{attribute 'monitoring' := 'call'}
PROPERTY INTERNAL PosHomeCh : LREAL
GET
PosHomeCh := stLocalSettings.stDynStationSettings[E_St010_Settings.eSt010_Settings_PosHomeCh].fValue;
END_GET
END_PROPERTY

{attribute 'monitoring' := 'call'}
PROPERTY INTERNAL PosWork : LREAL
GET
PosWork := stLocalSettings.stDynStationSettings[E_St010_Settings.eSt010_Settings_PosWork].fValue + // 1. Mitnehmerpos.
	  (OvenSegmentHeight * 
		TRUNC(((P_Plant.TrolleyRackDivision * stSt010IOvenA.iConfirmPosition) + 
		(OvenSegmentHeight - OvenFixPartHeight - 50))/OvenSegmentHeight)); // -50 => height axis z
END_GET
END_PROPERTY

{attribute 'monitoring' := 'call'}
PROPERTY INTERNAL PosWorkCh : LREAL
GET
PosWorkCh := stLocalSettings.stDynStationSettings[E_St010_Settings.eSt010_Settings_PosWorkCh].fValue;
END_GET
END_PROPERTY

{attribute 'monitoring' := 'call'}
PROPERTY INTERNAL PosWorkOpn : LREAL
GET
PosWorkOpn := PosWork + 

			  LMOD(((P_Plant.TrolleyRackDivision * stSt010IOvenA.iConfirmPosition) + (P_Plant.TrolleyRackOriginX - OvenFixPartHeight - 50)), 
					OvenSegmentHeight) + 
					50 + // -50 => height axis z
			  P_Plant.TrolleyRackDivision; // ( + TrolleyDevisionY --> safety distance)
END_GET
END_PROPERTY

/// Reset station logic
{attribute 'object_name' := 'Reset'}
METHOD Reset
VAR
END_VAR
// base logic run
SUPER^.Reset();

// reset objects
//diContinuesNok := 0;

IF fbAxis.bError OR NOT RunCycle THEN
	fbAxis.Reset();
END_IF
IF fbAxisCh1.bError OR NOT RunCycle THEN
	fbAxisCh1.Reset();
END_IF
IF fbAxisCh2.bError OR NOT RunCycle THEN
	fbAxisCh2.Reset();
END_IF
END_METHOD

{attribute 'monitoring' := 'call'}
PROPERTY PRIVATE WorkSpeed : LREAL
GET
WorkSpeed := stLocalSettings.stDynStationSettings[E_St010_Settings.eSt010_Settings_WorkSpeed].fValue;
END_GET
END_PROPERTY

{attribute 'monitoring' := 'call'}
PROPERTY PRIVATE WorkSpeedCh : LREAL
GET
WorkSpeedCh := stLocalSettings.stDynStationSettings[E_St010_Settings.eSt010_Settings_WorkSpeedCh].fValue;
END_GET
END_PROPERTY

END_FUNCTION_BLOCK

// ---- POUs/Components/AxisDriver/FB_Axis_Ui.TcPOU
/// Visu Interface für Achse
FUNCTION_BLOCK FB_Axis_Ui EXTENDS FB_ManualUiBase
VAR_INPUT
	///	Zus. Freigabe für Positive Richtung	
	bFreigabe_P		: BOOL := TRUE;
	///	Zus. Freigabe für Negative Richtung	
	bFreigabe_N		: BOOL := TRUE;
	
	/// Tippen +
	bJogP			:BOOL;
	/// Tippen -
	bJogN			:BOOL;
	/// GoTo
	//bGoTo		:BOOL;
	/// Geschwindigkeit
	fVelocity		:REAL := 1;
	
	/// Maximaler Weg pro Bewegung
	fMaxWeg			: REAL := 500;
	bModulo			: BOOL := FALSE;
	bEnableRefReset	: BOOL;	
	bEnableGear		: BOOL := FALSE;
	fGearRatio		: LREAL := 1;
	eMasterAxisId	: E_Axis := E_Axis.eAxis_none;
	bEnableBrakeControl	: BOOL := FALSE;
	bEnableSetPos	: BOOL := FALSE;
	
	// axis manager
	stAxisManager	: ST_AxisManager;
	stUnit			: ST_Text;
END_VAR
VAR_IN_OUT
	/// Achse in GRST
	bInHome			: BOOL;
	// axis reference
	fbAxis			: FB_AxisDriver;
	// hmi control IN
	stHMIControlIn	: ST_HMI_MANUAL_AXIS_IN;
	// hmi control OUT
	stHMIControlOut	: ST_HMI_MANUAL_AXIS_OUT;
END_VAR
VAR_OUTPUT	
	/// 0=Undefiniert; 
	/// 1=Fehler; 
	/// 2=Fahrt Positiv; 
	/// 3=Fahrt Negativ
	/// 4=Stillstand
	/// 5=Synchron
	iStatus				: INT;
	stState				: ST_Text;
	
	/// Servo Istposition
	fPosition			: LREAL;
	diColor_Position	: UDINT := STATICS.stColor.Gray;
	diColor_State		: UDINT;
	diColorSelectedItem	: UDINT;
	sText_State			: STRING;
END_VAR
VAR
	nn	: INT;
	stAxisState				: Tc2_MC2.ST_AxisStatus;
	eManualMode				: E_ManualMode;
	eManualModeOLD			: E_ManualMode;
	
	posEnableManual			: R_TRIG;
	negEnableManual			: F_TRIG;
	posIndexChanged			: R_TRIG;
	rtrigGearIn				: R_TRIG;
	ftrigGearOut			: F_TRIG;
	posGoTo,
	posGear,
	posTip_P,
	posTip_N,
	posRefReset,	
	rtrigTargetListClick,			
	rtrigBrake				: R_TRIG;
	
	fTargetPos				: LREAL;
	fStartPos				: LREAL;
	bManualModeAbsolute,
	bMovingAbs				: BOOL;
	bGear					: BOOL;
	
	bBrakeOff				: BOOL;
	
	posSelGoTo,
	posTippPos,
	posTippNeg,
	posSelJogTipp,
	posSelJog001,
	posSelJog01,
	posSelJog1,
	posSelJog10,
	posSelJog100,
	posSelMoveSollposAbs	: R_TRIG;
	
	tonRefReset				: TON;
	
	fSollPositionLatched	: REAL;
	
	stHomeParameter			: ST_AxisHomingParameter;
	
	tonTagetListClick		: ton;
	bTagetListClickSave		: BOOL;
	nTargetListIdx			: UINT;
	bFromTargetList			: BOOL; // FALSE from Input feld TRUE from List
	
	// master axis reference, if needed (else, set to dummy)
	stMasterAxisRef			: REFERENCE TO AXIS_REF REF= NcIO.stAxisDummy;
END_VAR
VAR PERSISTENT
	stTargetList			: ARRAY[0..9] OF ST_UserControl_Manual_Axis_Item; /// product data
	bCalibratedLocal		: BOOL;
END_VAR

(*
	Baustein zum bedienen einer Achse ueber die Visu
*)
stName := fbAxis.Name;
nTargetListIdx := stHMIControlIn.nSelectedRowIndex;
M_AxisManager();

IF (diObjectIndex = diSelectedObjectIndex) AND (diObjectIndex <> 0) AND bEnableManual THEN
	bManualActive := TRUE;
	stHMIControlOut.bVisible := TRUE;
	stHMIControlOut.bVisibleGear := bEnableGear;
	stHMIControlOut.bVisibleRefReset := bEnableRefReset;
	stHMIControlOut.bVisibleBrake := bEnableBrakeControl;
	stHMIControlOut.bVisibleSetPos := bEnableSetPos;
	stName:= stHMIControlOut.stObjectName := fbAxis.Name;

	stHMIControlOut.sOverride := SEL(fbAxis.bHoldActiv,LREAL_TO_FMTSTR(REAL_TO_LREAL(fbAxis.Override), 4, FALSE),'Hold Activ');
	stHMIControlOut.sTargetPosition := LREAL_TO_FMTSTR(REAL_TO_LREAL(fTargetPos), 4, FALSE);
	
	IF bModulo THEN
		stHMIControlOut.sActPosition := LREAL_TO_FMTSTR(fbAxis.ModuloPosition, 4, FALSE);
	ELSE
		stHMIControlOut.sActPosition := LREAL_TO_FMTSTR(fbAxis.Position, 4, FALSE);
	END_IF
	
	IF stAxisState.Coupled THEN
		stHMIControlOut.stGearStatus := F_CreateDynText("coupled", 0);
	ELSE
		stHMIControlOut.stGearStatus := F_CreateDynText("uncoupled", 0);
	END_IF
	
	IF NOT fbAxis.Homed THEN
		stHMIControlOut.stRefStatus := F_CreateDynText("unreferenced", 0);
	ELSE
		stHMIControlOut.stRefStatus := F_CreateDynText("referenced", 0);
	END_IF
	
	stHMIControlOut.stButtonGoTo.stName := CONST.stTextListGlobal.stText_GoTo;
	stHMIControlOut.stButtonJogPos.stName := CONST.stTextListGlobal.stText_JogPos;
	stHMIControlOut.stButtonJogNeg.stName := CONST.stTextListGlobal.stText_JogNeg;
	stHMIControlOut.stButtonGear.stName := CONST.stTextListGlobal.stText_Gear;
	stHMIControlOut.stButtonRefReset.stName := CONST.stTextListGlobal.stText_RefReset;
	stHMIControlOut.stButtonBrake.stName := CONST.stTextListGlobal.stText_Brake;
	stHMIControlOut.stButtonSetPos.stName := CONST.stTextListGlobal.stText_SetPos;

	stHMIControlOut.aJogModeName[0] :=  CONST.stTextListGlobal.stText_Jogpermanent;
	stHMIControlOut.aJogModeName[1] :=  CONST.stTextListGlobal.stText_Jog_0_01;
	stHMIControlOut.aJogModeName[2] :=  CONST.stTextListGlobal.stText_Jog_0_1;
	stHMIControlOut.aJogModeName[3] :=  CONST.stTextListGlobal.stText_Jog_1_0;	
	stHMIControlOut.aJogModeName[4] :=  CONST.stTextListGlobal.stText_Jog_10_0;	
	
	stHMIControlOut.stButtonGoTo.stColor.color := F_ColorToStringHexColor(STATICS.stColor.Theme);
	stHMIControlOut.stButtonJogPos.stColor.color := F_ColorToStringHexColor(STATICS.stColor.Theme);
	stHMIControlOut.stButtonJogNeg.stColor.color := F_ColorToStringHexColor(STATICS.stColor.Theme);
	stHMIControlOut.stButtonGear.stColor.color := F_ColorToStringHexColor(STATICS.stColor.Theme);
	stHMIControlOut.stButtonRefReset.stColor.color := F_ColorToStringHexColor(STATICS.stColor.Theme);
	stHMIControlOut.stButtonBrake.stColor.color := F_ColorToStringHexColor(STATICS.stColor.Theme);
	
	IF stHMIControlIn.stButtonGoTo.bClick AND bMovingAbs THEN
		stHMIControlOut.stButtonGoTo.stColor.color := F_ColorToStringHexColor(STATICS.stColor.LimeGreen);
	END_IF
	IF stHMIControlIn.stButtonJogPos.bClick AND NOT bMovingAbs AND fbAxis.Velocity > 0.5 THEN
		stHMIControlOut.stButtonJogPos.stColor.color := F_ColorToStringHexColor(STATICS.stColor.LimeGreen);
	END_IF
	IF stHMIControlIn.stButtonJogNeg.bClick AND NOT bMovingAbs AND fbAxis.Velocity < -0.5 THEN
		stHMIControlOut.stButtonJogNeg.stColor.color := F_ColorToStringHexColor(STATICS.stColor.LimeGreen);
	END_IF
	IF bGear THEN
		stHMIControlOut.stButtonGear.stColor.color := F_ColorToStringHexColor(STATICS.stColor.LimeGreen);
	END_IF
	IF tonRefReset.Q THEN
		stHMIControlOut.stButtonRefReset.stColor.color := F_ColorToStringHexColor(STATICS.stColor.LimeGreen);
	END_IF	
	IF bBrakeOff THEN
		stHMIControlOut.stButtonBrake.stColor.color := F_ColorToStringHexColor(STATICS.stColor.LimeGreen);
	END_IF	

	// Timer, Flanken
	posTip_P(CLK := bJogP OR stHMIControlIn.stButtonJogPos.bClick);
	posTip_N(CLK := bJogN OR stHMIControlIn.stButtonJogNeg.bClick);
	posGoTo(CLK := (*bGoTo OR*) stHMIControlIn.stButtonGoTo.bClick);
	posGear(CLK := stHMIControlIn.stButtonGear.bClick);
	rtrigTargetListClick(CLK := stHMIControlIn.bSetTargetFromList);
	tonRefReset.PT := T#1S;
	tonRefReset.IN := stHMIControlIn.stButtonRefReset.bClick;
	tonRefReset();
	posRefReset(CLK := tonRefReset.Q);	
	rtrigBrake(CLK := stHMIControlIn.stButtonBrake.bClick); 
	IF posTip_N.Q OR posTip_P.Q THEN
		bMovingAbs := FALSE;
		bManualModeAbsolute := FALSE;
	ELSIF posGoTo.Q THEN
		bManualModeAbsolute := TRUE;
	END_IF
	IF posGear.Q AND fbAxis.NotMoving THEN
		bGear := NOT bGear;
	END_IF
	IF rtrigBrake.Q AND (fbAxis.NotMoving OR TRUE)THEN
		bBrakeOff := NOT bBrakeOff;
	END_IF
ELSE
	IF bManualActive THEN
		bManualActive := FALSE;
		stHMIControlOut.bVisible := FALSE;
	END_IF
	bBrakeOff := FALSE;
END_IF	
	
// nicht aktiv -> alles löschen und Exit
IF NOT fbAxis.Active THEN
	bError := FALSE ;
	stErrorText := CONST.stTextListGlobal.stText_notext;
	iStatus := 0;// 0=Undefiniert
	fPosition := 0;
	A_StateMapping();
	RETURN;
END_IF

// Object mit Index ausgewählt
IF (diObjectIndex = diSelectedObjectIndex) THEN
	diColorSelectedItem := STATICS.stColor.LimeGreen;
ELSE
	diColorSelectedItem := STATICS.stColor.Gray;
END_IF

bError := fbAxis.State = E_ComponentState.eComponentState_error;
IF bError THEN
	stErrorText := F_CreateDynTextDefault(fbAxis.ClearText);
ELSE
	stErrorText := CONST.stTextListGlobal.stText_notext;
END_IF
fPosition := fbAxis.Position; // Istposition der Achse

// Status
stAxisState := fbAxis.AxisState;
IF bError THEN
	iStatus := 1; // 1=Fehler; 
	diColor_State:= STATICS.stColor.Red;
	stState.wsNameId := "error";
	stState.wsName := "error";
	stState.nNameId :=1;
ELSIF stAxisState.Moving AND stAxisState.PositiveDirection THEN
	iStatus := 2; // 2=Fahrt Positiv; 
	diColor_State:= STATICS.stColor.Green;
	stState.wsNameId := "movepositive";
	stState.wsName := "movepositive";
	stState.nNameId :=2;
ELSIF stAxisState.Moving AND stAxisState.NegativeDirection THEN
	iStatus := 3; // 3=Fahrt Negativ;
	diColor_State:= STATICS.stColor.Green;
	stState.wsNameId := "movenegative";
	stState.wsName := "movenegative";
	stState.nNameId :=3;
ELSIF stAxisState.Coupled THEN
	iStatus := 5; // 5=Synchron
	diColor_State:= STATICS.stColor.LightSkyBlue;
	stState.wsNameId := "coupled";
	stState.wsName := "coupled";
	stState.nNameId :=5;
ELSIF NOT stAxisState.Moving THEN
	iStatus := 4; // 4=Stillstand
	diColor_State:= STATICS.stColor.Gray;
	stState.wsNameId := "notmoveing";
	stState.wsName := "notmoveing";
	stState.nNameId :=4;
ELSE
	iStatus := 0;// 0=Undefiniert
	diColor_State:= STATICS.stColor.Orange;
	stState.wsNameId := "undifined";
	stState.wsName := "undifined";
	stState.nNameId :=0;
END_IF

//Statuszahl Text Zuweisung
CASE iStatus OF
	0:
		sText_State := ('Undefiniert');
	1:
		sText_State := ('Fehler');
	2:
		sText_State := ('Fahrt Positiv');
	3:
		sText_State := ('Fahrt Negativ');
	4:
		sText_State := ('Stillstand OK');
	5:
		sText_State := ('Synchron');
END_CASE

bWarning := FALSE;
stWarnText := CONST.stTextListGlobal.stText_notext;

// Achse stoppen bei Umschaltung(en)
posEnableManual(CLK := bEnableManual);
negEnableManual(CLK := bEnableManual);
posIndexChanged(CLK := bEnableManual AND (diObjectIndex <> diSelectedObjectIndex));
IF posEnableManual.Q OR negEnableManual.Q OR posIndexChanged.Q THEN
	IF fbAxis.Moving THEN
		fbAxis.Halt();
	END_IF
	bMovingAbs := FALSE;
END_IF

// Homing Zurücksetzen
IF posRefReset.Q AND fbAxis.NotMoving AND fbAxis.Homed AND bEnableRefReset THEN
	stHomeParameter.eHomingMode := MC_HomingMode.MC_ResetCalibration;
	fbAxis.HomeEx(stHomeParameter);
END_IF

// exit wenn nicht dieses Objekt
IF NOT bEnableManual OR (diObjectIndex <> diSelectedObjectIndex) THEN
	bMovingAbs := FALSE;
	A_StateMapping();
	RETURN;
END_IF


// Handbedienlogik
// werwenden von Handbediencontrol direkt
// Status wird in diesem FB gemerkt und wiedereingestellt

// Auswahl Manuelle Funktionen
A_SelectManualMode();

// Modus wurde geändert -> Achse stoppen
IF eManualMode <> eManualModeOLD THEN
	eManualModeOLD := eManualMode;
	IF fbAxis.Moving THEN
		fbAxis.Halt();
	END_IF
	bMovingAbs := FALSE;
	bBrakeOff := FALSE;
END_IF

// Bei Stillstand und Taste Gear in HMI Koppeln
rtrigGearIn(CLK := bGear);
ftrigGearOut(CLK := bGear);
IF fbAxis.NotMoving AND rtrigGearIn.Q AND bEnableGear THEN
	fbAxis.GearIn(fGearRatio, eMasterAxisId, stMasterAxisRef);
END_IF
IF fbAxis.NotMoving AND ftrigGearOut.Q THEN
	fbAxis.GearOut();
END_IF

//Bremsen Steuerung
IF fbAxis.bHasJob OR NOT bEnableBrakeControl THEN
	bBrakeOff := FALSE;
END_IF
IF bBrakeOff THEN
	; //todo brake control
END_IF

FOR nn := 0 TO 9 DO
	stHMIControlout.stTargetList[nn].stName := stTargetList[nn].stName;
	stHMIControlout.stTargetList[nn].stPos.wsNameId := stHMIControlout.stTargetList[nn].stPos.wsName := TO_WSTRING(stTargetList[nn].fPos);
END_FOR

//set Target from Target List
fTargetPos := SEL(bFromTargetList AND nTargetListIdx >= 0 AND nTargetListIdx <= 9, 
					stHMIControlIn.fTargetPosition, 
					stTargetList[nTargetListIdx].fPos);

IF rtrigTargetListClick.Q THEN
	bTagetListClickSave := TRUE;
END_IF

tonTagetListClick(IN := bTagetListClickSave, PT := T#1S);
IF tonTagetListClick.Q THEN
	bTagetListClickSave := FALSE;
	IF (stTargetList[nTargetListIdx].stName.wsNameId <> "") OR (stTargetList[nTargetListIdx].stName.wsName <> "") THEN
		bFromTargetList := TRUE;
	END_IF
END_IF
IF stHMIControlIn.bSetTarget THEN
	bFromTargetList := FALSE;	
END_IF

// Manuelle Bewegungen
// Tippen konstant
IF (eManualMode = E_ManualMode.eManualMode_Tippen) THEN
	IF posTip_P.Q OR posTip_N.Q THEN
		bInHome := FALSE;
		fStartPos := fbAxis.Position;
	END_IF
	fbAxis.JogExVel(((bJogN OR stHMIControlIn.stButtonJogNeg.bClick) AND bFreigabe_N), 	// Tip N, max Weg		ABS(fbAxis.Position - fStartPos) < fMaxWeg
					((bJogP OR stHMIControlIn.stButtonJogPos.bClick) AND bFreigabe_P), 	// Tip P, max Weg		ABS(fbAxis.Position - fStartPos) < fMaxWeg)
					fVelocity/2, E_JogMode.MC_JOGMODE_CONTINOUS);
					
// Tippen um 0.01 Einheit
ELSIF (eManualMode = E_ManualMode.eManualMode_Jog001) THEN
	IF posTip_P.Q AND bFreigabe_P THEN
		bInHome := FALSE;
		fbAxis.MoveRelExVel(0.01, fVelocity);
	END_IF
	IF posTip_N.Q AND bFreigabe_N THEN
		bInHome := FALSE;
		fbAxis.MoveRelExVel(-0.01, fVelocity);
	END_IF					

// Tippen um 0.1 Einheit
ELSIF (eManualMode = E_ManualMode.eManualMode_Jog01) THEN
	IF posTip_P.Q AND bFreigabe_P THEN
		bInHome := FALSE;
		fbAxis.MoveRelExVel(0.1, fVelocity);
	END_IF
	IF posTip_N.Q AND bFreigabe_N THEN
		bInHome := FALSE;
		fbAxis.MoveRelExVel(-0.1, fVelocity);
	END_IF

// Tippen um 1 Einheit
ELSIF (eManualMode = E_ManualMode.eManualMode_Jog1) THEN
	IF posTip_P.Q AND bFreigabe_P THEN
		bInHome := FALSE;
		fbAxis.MoveRelExVel(1.0, fVelocity);
	END_IF
	IF posTip_N.Q AND bFreigabe_N THEN
		bInHome := FALSE;
		fbAxis.MoveRelExVel(-1.0, fVelocity);
	END_IF

// Tippen um 10 Einheiten
ELSIF (eManualMode = E_ManualMode.eManualMode_Jog10) THEN
	IF posTip_P.Q AND bFreigabe_P THEN
		bInHome := FALSE;
		fbAxis.MoveRelExVel(10.0, fVelocity);
	END_IF
	IF posTip_N.Q AND bFreigabe_N THEN
		bInHome := FALSE;
		fbAxis.MoveRelExVel(-10.0, fVelocity);
	END_IF

// Tippen um 100 Einheiten
(*ELSIF (eManualMode = E_ManualMode.eManualMode_Jog100) THEN
	IF posTip_P.Q AND bFreigabe_P THEN
		fbAxis.MoveRelExVel(100.0, fVelocity);
	END_IF
	IF posTip_N.Q AND bFreigabe_N THEN
		fbAxis.MoveRelExVel(-100.0, fVelocity);
	END_IF	*)
END_IF

// Position anfahren solange Tip Taste gedrueckt
IF bManualModeAbsolute THEN //IF (eManualMode = E_ManualMode.eManualMode_MoveSollAbs) THEN

	// Halt	
	IF NOT stHMIControlIn.stButtonGoTo.bClick THEN//bGoTo THEN
		IF fbAxis.Moving THEN
			fbAxis.Halt();
		END_IF
		fSollPositionLatched := fTargetPos;//stVisuControlPanel.fSollPosition;
		bMovingAbs := FALSE;
		
	// los
	// Start oder Soll Position geändert
	ELSIF posGoTo.Q OR (fbAxis.Moving AND fSollPositionLatched <> fTargetPos(*stVisuControlPanel.fSollPosition*)) THEN
		fSollPositionLatched := fTargetPos;//stVisuControlPanel.fSollPosition;
		fStartPos := fbAxis.Position;
		bMovingAbs := TRUE;
		
		// möchte in Positive Richtung fahren, keine Freigabe = Alarm
		IF ((*stVisuControlPanel.fSollPosition*)fTargetPos > fbAxis.Position) THEN
			IF bFreigabe_P THEN
				IF NOT bModulo THEN
					fbAxis.MoveAbsExVel(fTargetPos(*stVisuControlPanel.fSollPosition*), fVelocity);
				ELSE
					fbAxis.MoveModExVel(fTargetPos(*stVisuControlPanel.fSollPosition*), fVelocity);
				END_IF
				bInHome := FALSE;
			ELSE
				bWarning := TRUE;
				stWarnText := CONST.stTextListGlobal.stText_Comp.stText_AxisUi_PosDirectionWarn;				
			END_IF
			
		// möchte in Negative Richtung fahren, keine Freigabe = Alarm
		ELSIF ((*stVisuControlPanel.fSollPosition*)fTargetPos < fbAxis.Position) THEN
			IF bFreigabe_N THEN
				IF NOT bModulo THEN
					fbAxis.MoveAbsExVel(fTargetPos(*stVisuControlPanel.fSollPosition*), fVelocity);	
				ELSE
					fbAxis.MoveModExVel(fTargetPos(*stVisuControlPanel.fSollPosition*), fVelocity);	
				END_IF		
				bInHome := FALSE;
			ELSE
				bWarning := TRUE;
				stWarnText := CONST.stTextListGlobal.stText_Comp.stText_AxisUi_NegDirectionWarn;				
			END_IF
			
		END_IF
		
	// max. Weg Begrenzen
	ELSIF (ABS(fbAxis.Position - fStartPos) > fMaxWeg) AND fbAxis.Moving AND bMovingAbs THEN
		fbAxis.Halt();
		bMovingAbs := FALSE;
	END_IF
	
END_IF


//IF (eManualMode <> E_ManualMode.eManualMode_MoveSollAbs) THEN
//	bMovingAbs := FALSE;
//END_IF

A_StateMapping();

ACTION A_SelectManualMode:

// Auswahl Manuelle Funktionen

posSelGoTo(CLK := stHMIControlIn.stButtonGoTo.bClick);
posTippPos(CLK := stHMIControlIn.stButtonJogPos.bClick);
posTippNeg(CLK := stHMIControlIn.stButtonJogNeg.bClick);

CASE stHMIControlIn.eJogMode OF
	E_Axis_JogMode.eJogMode_0: // Tippen um Schritt
		eManualMode := E_ManualMode.eManualMode_Tippen;
	E_Axis_JogMode.eJogMode_1: // Tippen um 0,01
		eManualMode := E_ManualMode.eManualMode_Jog001;
	E_Axis_JogMode.eJogMode_2: // Tippen um 0,1
		eManualMode := E_ManualMode.eManualMode_Jog01;
	E_Axis_JogMode.eJogMode_3: // Tippen um 1
		eManualMode := E_ManualMode.eManualMode_Jog1;
	E_Axis_JogMode.eJogMode_4: // Tippen um 10
		eManualMode := E_ManualMode.eManualMode_Jog10;
	E_Axis_JogMode.eJogMode_5: // Tippen um 100
		eManualMode := E_ManualMode.eManualMode_Jog100;
	//E_Axis_JogMode.eJogMode_1: // Absolut Positionieren
	//	eManualMode := E_ManualMode.eManualMode_MoveSollAbs;	
END_CASE

//posSelJogTipp(CLK := stVisuControlPanel.bTippen);
//posSelJog001(CLK := stVisuControlPanel.bJog001);
//posSelJog01(CLK := stVisuControlPanel.bJog01);
//posSelJog1(CLK := stVisuControlPanel.bJog1);
//posSelJog10(CLK := stVisuControlPanel.bJog10);
//posSelJog100(CLK := stVisuControlPanel.bJog100);
//posSelMoveSollposAbs(CLK := stVisuControlPanel.bSollposAnfahren);

//IF posSelJogTipp.Q THEN
//	eManualMode := E_ManualMode.eManualMode_Tippen;
//END_IF
//IF posSelJog001.Q THEN
//	eManualMode := E_ManualMode.eManualMode_Jog001;
//END_IF
//IF posSelJog01.Q THEN
//	eManualMode := E_ManualMode.eManualMode_Jog01;
//END_IF
//IF posSelJog1.Q THEN
//	eManualMode := E_ManualMode.eManualMode_Jog1;
//END_IF
//IF posSelJog10.Q THEN
//	eManualMode := E_ManualMode.eManualMode_Jog10;
//END_IF
//IF posSelJog100.Q THEN
//	eManualMode := E_ManualMode.eManualMode_Jog100;
//END_IF
//IF posSelMoveSollposAbs.Q THEN
//	eManualMode := E_ManualMode.eManualMode_MoveSollAbs;
//END_IF

//// andere Typen
//stVisuControlPanelStatus.bAusSelected := FALSE;
//stVisuControlPanelStatus.bEinSelected := FALSE;
//// Servos
/////Servo Tippen	
//stVisuControlPanelStatus.bTippenSelected := (eManualMode = E_ManualMode.eManualMode_Tippen);
/////Servo Jog 0.01
//stVisuControlPanelStatus.bJog001Selected := (eManualMode = E_ManualMode.eManualMode_Jog001);
/////Servo Jog 0.1
//stVisuControlPanelStatus.bJog01Selected := (eManualMode = E_ManualMode.eManualMode_Jog01);
/////Servo Jog 1
//stVisuControlPanelStatus.bJog1Selected := (eManualMode = E_ManualMode.eManualMode_Jog1);
/////Servo Jog 10
//stVisuControlPanelStatus.bJog10Selected := (eManualMode = E_ManualMode.eManualMode_Jog10);
/////Servo Jog 100
//stVisuControlPanelStatus.bJog100Selected := (eManualMode = E_ManualMode.eManualMode_Jog100);
/////Servo Sollposition Anfahren
//stVisuControlPanelStatus.bSollposAnfahrenSelected := (eManualMode = E_ManualMode.eManualMode_MoveSollAbs);
END_ACTION

ACTION A_StateMapping:
IF NOT __ISVALIDREF(stStateObject) THEN
	RETURN;
END_IF

// state mapping
stStateObject.stState := stState;
stStateObject.stValue.wsName := TO_WSTRING(LREAL_TO_FMTSTR(REAL_TO_LREAL(fPosition), 2, FALSE));
stStateObject.nIndexColor := diColorSelectedItem;
END_ACTION

METHOD PRIVATE M_AxisManager : BOOL
VAR_INPUT
END_VAR
// map axis info
stAxisManager.bAxisEnabled := fbAxis.bEnable;
stAxisManager.bCalibrated := SEL(stAxisManager.bUseLocalCalibration, fbAxis.Homed, bCalibratedLocal);
stAxisManager.fActPos := fbAxis.Position;
stAxisManager.stBmk := stBmk;
stAxisManager.stName := stName;
stAxisManager.stUnit := stUnit;
//stAxisManager.stInfo := ST_Text;

// set/reset calibration
IF stAxisManager.bSetCalibration THEN
	stAxisManager.bSetCalibration := FALSE;
	IF stAxisManager.bUseLocalCalibration THEN bCalibratedLocal := TRUE; RETURN; END_IF
	fbAxis.SetCalibration(TRUE);
ELSIF stAxisManager.bResetCalibration THEN
	stAxisManager.bResetCalibration := FALSE;
	IF stAxisManager.bUseLocalCalibration THEN bCalibratedLocal := FALSE; RETURN; END_IF
	fbAxis.SetCalibration(FALSE);
END_IF

// set ax pos offset
IF stAxisManager.bSetPosGo THEN
	stAxisManager.bSetPosGo := FALSE;
	fbAxis.SetAxPosOffs(stAxisManager.fSetPos);
END_IF
END_METHOD

METHOD PUBLIC M_SetMaserAxRef : BOOL
VAR_IN_OUT
	fbAxRef : AXIS_REF;
END_VAR
stMasterAxisRef REF= fbAxRef;
END_METHOD

METHOD PUBLIC M_TargetListAddItem : BOOL
VAR_INPUT
	stSetName		: ST_Text;
	fSetPosition	: LREAL;
END_VAR
FOR nn := 0 TO 9 DO
	IF (stTargetList[nn].stName.wsNameId = stSetName.wsNameId)OR (stTargetList[nn].stName.wsName = stSetName.wsName)THEN
		stTargetList[nn].fPos := fSetPosition;
		EXIT;
	ELSIF (stTargetList[nn].stName.wsNameId = "") AND (stTargetList[nn].stName.wsName = "") THEN
		stTargetList[nn].stName := stSetName;
		stTargetList[nn].fPos := fSetPosition;
		EXIT;
	END_IF
END_FOR
END_METHOD

METHOD M_TargetListClear : BOOL
VAR_INPUT
END_VAR
MEMSET(ADR(stTargetList), 0, SIZEOF(stTargetList));
END_METHOD

PROPERTY ManualMode : E_ManualMode
GET
ManualMode := eManualMode;
END_GET
SET
eManualMode := ManualMode;
END_SET
END_PROPERTY

END_FUNCTION_BLOCK

// ---- POUs/Components/FurnaceDriver/FB_FurnaceDriver.TcPOU
/// Exhaustion driver.
FUNCTION_BLOCK FB_FurnaceDriver EXTENDS FB_ComponentBase

VAR CONSTANT
	nFurnanceScheduleItems		: INT := 7;
END_VAR

VAR
	/// IO structure
	stIn 				: REFERENCE TO ST_FurnaceIn;
	stOut 				: REFERENCE TO ST_FurnaceOut;
	
	/// fb
	fbTmpCtrl			: FB_CTRL_TempController;
	
	/// Sequences
	eSequenceId			: E_FurnaceSeq;
	
	nStep				: INT;
	
	// private var's
	stCTRLParameter		: ST_CTRL_TempCtrlParameter;
	stPIDParameter		: ST_CTRL_ParaController;
	
	fTemperature		: LREAL;
	fSlope				: LREAL;
	fInitial			: LREAL;
	bkpAlarmSupp		: DWORD;	
	eCTRL_Mode 			: E_CTRL_MODE := E_CTRL_MODE.eCTRL_MODE_IDLE; 	(*   eCTRL_MODE_TUNE  ;*)
	bTuned				: BOOL;	
	rtOverheat			: R_TRIG;

END_VAR

///
/// Furnace driver.
/// Hannes Fuger / asma.at / 12.2015
///

METHOD PRIVATE _AUTO 
VAR_INPUT
END_VAR
CASE nStep OF
	
0	:	// switch to Active mode
		eCTRL_Mode := E_CTRL_MODE.eCTRL_MODE_ACTIVE;
		stCtrlParameter.bSelCtrlParameterSet := TRUE;
						
		IF fbTmpCtrl.eCtrlState = e_Ctrl_state.eCTRL_STATE_ACTIVE THEN
			nStep := 99;
		END_IF			


END_CASE
END_METHOD

METHOD _HAND
VAR_INPUT
END_VAR
CASE nStep OF
	
0	:	// switch to Active mode
		eCTRL_Mode := E_CTRL_MODE.eCTRL_MODE_MANUAL;
		stCtrlParameter.bSelCtrlParameterSet := TRUE;
							
		IF fbTmpCtrl.eCtrlState = e_Ctrl_state.eCTRL_STATE_MANUAL THEN
			nStep := 99;
		END_IF	
		
END_CASE
END_METHOD

METHOD _OFF
VAR_INPUT
END_VAR
CASE nStep OF
	
0	:	// switch to Active mode
		eCTRL_Mode := E_CTRL_MODE.eCTRL_MODE_IDLE;
							
		IF fbTmpCtrl.eCtrlState = e_Ctrl_state.eCTRL_STATE_IDLE THEN
			nStep := 99;
		END_IF	
			
END_CASE
END_METHOD

METHOD _TUNE
VAR_INPUT
END_VAR
CASE nStep OF
	
0	:	// switch to Tune mode
		eCTRL_Mode := E_CTRL_MODE.eCTRL_MODE_TUNE;
		// Alarme ausstellen
		bkpAlarmSupp := stCTRLParameter.dwAlarmSupp;
		stCtrlParameter.bSelCtrlParameterSet := FALSE;
		
		IF fbTmpCtrl.eCtrlState = e_Ctrl_state.eCTRL_STATE_TUNING THEN
			nStep := 10;
		END_IF

10	:	IF fbTmpCtrl.eCtrlState = e_Ctrl_state.eCTRL_STATE_TUNED THEN
			nStep := 20;
		END_IF
			
20	:	stPIDParameter := fbTmpCtrl.sParaControllerInternal;
		stCtrlParameter.bSelCtrlParameterSet := TRUE;
		fbTmpCtrl.eCtrlMode := E_CTRL_MODE.eCTRL_MODE_PASSIVE;
		eSequenceId := eFurnaceSeq_none;
		

END_CASE
END_METHOD

PROPERTY CtrlParameter : REFERENCE TO ST_CTRL_TempCtrlParameter
GET
ctrlParameter REF= stCTRLParameter;
END_GET
SET
stCTRLParameter := ctrlParameter;
END_SET
END_PROPERTY

PROPERTY CtrlState : E_CTRL_STATE
GET
CtrlState := fbTmpCtrl.eCtrlState;
END_GET
END_PROPERTY

PROPERTY Error : BOOL
GET
Error := fbTmpCtrl.bError;
END_GET
END_PROPERTY

PROPERTY ErrorId : E_CTRL_ERRORCODES
GET
ErrorId := fbTmpCtrl.eErrorId;
END_GET
END_PROPERTY

METHOD FB_init : BOOL
VAR_INPUT
	bInitRetains : BOOL; // if TRUE, the retain variables are initialized (warm start / cold start)
	bInCopyCode : BOOL;  // if TRUE, the instance afterwards gets moved into the copy code (online change)
END_VAR
eTyp := E_ComponentType.eComponentType_Furnace;
END_METHOD

PROPERTY Heating : E_HeatingState
GET
Heating := E_HeatingState.eHeatingState_none;

IF Mode = eFurnaceSeq_Auto AND ((NOT SelPointAutoTwo AND SetPointAuto <> 0) OR (SelPointAutoTwo AND SetPointAutoTwo <> 0)) THEN
	Heating := E_HeatingState.eHeatingState_on;	
ELSIF  Mode = eFurnaceSeq_Hand AND SetPointManual <> 0 THEN
	Heating := E_HeatingState.eHeatingState_on;
ELSE
	Heating := E_HeatingState.eHeatingState_off;	
END_IF
END_GET
END_PROPERTY

METHOD HeatingMode
VAR_INPUT
	eMode				: E_FurnaceSeq;
END_VAR
eSequenceId := eMode;
nStep := 0;
END_METHOD

METHOD LoadCtrlParam
VAR_INPUT
END_VAR
//stCtrlParameter	:= CtrlParameter;
	
(* general parameters ***************************************************************)
stCtrlParameter.iMode					:= 1										;	(* 1=heating, 2=cooling, 3=heating&cooling *)
stCtrlParameter.iReactionOnFailure		:= eCTRL_ReactionOnFailure_NoFailure	;	(* 0=controller off, 1=manual op, 2=yMin, 3=yMax *)

stCtrlParameter.bSelCtrlParameterSet	:= FALSE									;	(* FALSE = internal set, TRUE = external set *)
	                                                                                
stCtrlParameter.dwAlarmSupp				:= 16#0000EFFF								;	(* alarm suppression *)
stCtrlParameter.tCtrlCycleTime			:= T#1000MS									;	(* controller cycle time *)
stCtrlParameter.tTaskCycleTime			:= T#10MS									;	(* plc task cycle time *)
		                                                                            
(* tuning parameters ****************************************************************)         
stCtrlParameter.iTuningMode				:= 1										;	(* only heating, only cooling, first heating then cooling or vice versa *)
	                                                                                
stCtrlParameter.tTuneStabilisation		:= T#20S									;	(* wait for a stable system *)
	                                                                                
stCtrlParameter.fEndTunePercentHeating	:= 80.0										;	(* switch to closed loop control when X > 0.8*W *)
stCtrlParameter.fYTuneHeating			:= 100.0									;	(* step change while tuning operation *)
stCtrlParameter.fYStableHeating			:= 0.0										;	(* tuning operation *)
	                                                                                
stCtrlParameter.fEndTunePercentCooling	:= 20.0										;	(* switch to closed loop control when X < 0.2*W *)
stCtrlParameter.fYTuneCooling			:= 0.0										;	(* step change while tuning operation *)
stCtrlParameter.fYStableCooling			:= 0.0										;	(* tuning operation *)
stCtrlParameter.fScalingFactor			:= 1.0										;	(* Scaling factor for KP heating/cooling *)
		                                                                            
(* setpoint parameters **************************************************************)         
stCtrlParameter.fWMin					:= 0.0										;	(* lower limit *)
stCtrlParameter.fWMax					:= 200.0									;	(* upper limit *)
	                                                                                
(* start up *************************************************************************)                                                                      
stCtrlParameter.bEnableSoftStart		:= FALSE									;	(* FALSE = no soft start, TRUE = soft start *)
stCtrlParameter.bEnableRamping			:= FALSE									;	(* FALSE = no ramping, TRUE = ramping *)
	                                                                                
stCtrlParameter.fWStartUp				:= 0.0										;	(* soft start plateau setpoint *)
stCtrlParameter.tStartUp				:= T#0MS									;	(* soft start waiting time*)
stCtrlParameter.bStartUpRamping			:= FALSE									;	(* enable ramping while start up phase *)
stCtrlParameter.fWStartUpVeloPos		:= 1.0										;	(* max gradient for increasing setpoint in start up phase*)
stCtrlParameter.fWStartUpVeloNeg		:= 1.0										;	(* max gradient for decreasing setpoint in start up phase *)
	                                                                                
stCtrlParameter.fWVeloPos				:= 1.0										;	(* max gradient for increasing setpoint *)
stCtrlParameter.fWVeloNeg				:= 1.0										;	(* max gradient for decreasing setpoint *)	
	                                                                                
(* actual value parameters **********************************************************)         
stCtrlParameter.bFilter 				:= FALSE                                    ;
stCtrlParameter.tFilter					:= T#0S                                     ;
		                                                                            
(* deadband parameters **************************************************************)         
stCtrlParameter.bDeadband				:= FALSE                                    ;
stCtrlParameter.fEDeadband				:= 0.0										;	
		                                                                            
(* control value parameters *********************************************************)         
stCtrlParameter.fYMin					:= 0.0										;	(* lower limit *)
stCtrlParameter.fYMax					:= 100.0									;	(* upper limit *)
stCtrlParameter.fYManual				:= 0.0									 	;	(* manual operation*)
stCtrlParameter.fYOnFailure				:= 0.0										;	(* control value on failure *)
	                                                                                ;
stCtrlParameter.tPWMCycleTime			:= T#5S										;	(* PWM: period *)
stCtrlParameter.tPWMMinOffTime			:= T#0S										;	(* PWM: min off time *)
stCtrlParameter.tPWMMinOnTime			:= T#0S										;	(* PWM: min on time *)
stCtrlParameter.tPWMWaitingTime			:= T#0S										;	(* PWM: min waiting time *) (* not yet implemented !!!!*)
	                                                                                
stCtrlParameter.fYThresholdOff			:= 0.0										;	(* 3-Point: Off threshold *)
stCtrlParameter.fYThresholdOn			:= 0.0										;	(* 3-Point: On threshold *)
	                                                                                
stCtrlParameter.nCyclesForSwitchOver	:= 100                                      ;
	                                                                                
(* controller settings **************************************************************)         
stCtrlParameter.bEnablePreController 	:= FALSE									;	(* enable precontroller *)
stCtrlParameter.bEnableZones 			:= FALSE									;	(* enable zone around setpoint with open loop control *)
stCtrlParameter.bEnableCVFilter 		:= FALSE									;	(* enable filter for CV (type see iFilterType) *)
stCtrlParameter.iFilterType 			:= eCTRL_FilterType_FIRSTORDER			 	;	(* filtertype of CV filter *)
stCtrlParameter.iControllerType 		:= eCTRL_ControllerType_PID					;	(* used controller normally PID *)
			
(* min max temperatures	*************************************************************)
stCtrlParameter.TempLow					:= -5.0										;
stCtrlParameter.TempLowLow				:= -10.0                                    ;
stCtrlParameter.TempHigh				:= 5.0                                      ;
stCtrlParameter.TempHighHigh			:= 10.0                                     ;
stCtrlParameter.TempAbsoluteHigh		:= 200.0                                    ;
stCtrlParameter.TempAbsoluteLow			:= 0.0	                                    ;
		                                                                            
(* internal tuning parameters *******************************************************)                                                    
stCtrlParameter.fTuneKp					:= 0.5                                      ;
stCtrlParameter.fTuneTn					:= 3                                     	;
stCtrlParameter.fTuneTv					:= 1                                     	;
stCtrlParameter.fTuneTd					:= 0.25                                     ;
END_METHOD

PROPERTY Mode : E_FurnaceSeq
GET
IF  (nStep = 99) THEN
	Mode := eSequenceId;
ELSE
	Mode := E_FurnaceSeq.eFurnaceSeq_none;
END_IF
END_GET
END_PROPERTY

PROPERTY PIDParameter : REFERENCE TO ST_CTRL_ParaController
GET
PIDParameter REF= stPIDParameter;
END_GET
SET
stPIDParameter := PIDParameter;
END_SET
END_PROPERTY

/// Reset component logic
{attribute '' := ''}
{attribute 'object_name' := 'Reset'}
METHOD Reset

VAR
	eOldMode			: E_FurnaceSeq;
END_VAR
// base logic run
SUPER^.Reset();

eSequenceId := E_FurnaceSeq.eFurnaceSeq_none;
nStep := 0;
END_METHOD

/// Run component logic
{attribute 'object_name' := 'Run'}
METHOD Run : E_ComponentState
VAR
	CtrlParameter			: ST_CTRL_TempCtrlParameter;
END_VAR
// base logic run
Run := SUPER^.Run();

// Sequencer 
SeqRun();

// convert Temperature
fTemperature := fSlope * INT_TO_LREAL(stIn.nTemperature) + fInitial;

// TemperatureCtrl
fbTmpCtrl(
		eCtrlMode				:= eCTRL_Mode, 
		//bSelSetpoint			:= FALSE, 
		//fW1						:= 120, 
		//fW2						:= 120, 
		fX						:= fTemperature, 
		//fYManual				:= , 
		bOpenThermocouple		:= FALSE, 
		bReverseThermocouple	:= FALSE, 
		bBackVoltage			:= FALSE, 
		bLeakage				:= FALSE, 
		bShortCircuit			:= FALSE, 
		bOpenCircuit			:= FALSE, 
		sParaControllerExternal	:= stPIDParameter, 
		sControllerParameter	:= stCTRLParameter, 
		);

// Analog output		
stOut.bPWMSignal := fbTmpCtrl.bYPWMPos;

// Choose set of controller parameters
//IF fbTmpCtrl.eCtrlState = eCTRL_STATE_TUNED THEN
//	eCTRL_Mode := eCTRL_MODE_ACTIVE;	
//END_IF

IF fbTmpCtrl.eCtrlState = e_Ctrl_state.eCTRL_STATE_ERROR THEN
	// todo: error
END_IF

rtOverheat.CLK := NOT stin.bOverheat;
rtOverheat();		

IF rtOverheat.Q THEN
//	WriteError(E_Event.eEvent_none, CONCAT(sName, ': Überhitzungsschutz'));
END_IF
END_METHOD

PROPERTY SelPointAutoTwo : BOOL
GET
SelPointAutoTwo := fbTmpCtrl.bSelSetpoint;
END_GET
SET
fbTmpCtrl.bSelSetpoint := SelPointAutoTwo;
END_SET
END_PROPERTY

METHOD SeqRun
VAR_INPUT
END_VAR

CASE eSequenceId OF

	eFurnaceSeq_hand:
		THIS^._HAND();
		
	eFurnaceSeq_auto:
		THIS^._AUTO();
	
	eFurnaceSeq_tune:
		THIS^._TUNE();
		
	eFurnaceSeq_off:
		THIS^._OFF();
END_CASE
END_METHOD

PROPERTY SetPointAuto : LREAL
GET
SetPointAuto := fbTmpCtrl.fW1;
END_GET
SET
fbTmpCtrl.fW1 := SetPointAuto;
END_SET
END_PROPERTY

PROPERTY SetPointAutoTwo : LREAL
GET
SetPointAutoTwo := fbTmpCtrl.fW2;
END_GET
SET
fbTmpCtrl.fW2 := SetPointAutoTwo;
END_SET
END_PROPERTY

PROPERTY SetPointManual : LREAL
GET
SetPointManual := fbTmpCtrl.fYManual;
END_GET
SET
fbTmpCtrl.fYManual := SetPointManual;
END_SET
END_PROPERTY

/// Set IO reference
{attribute 'object_name' := 'SetReferences'}
METHOD SetReferences
VAR_IN_OUT
	/// IO structure
	stRefIO 	: ST_FurnaceIO;
END_VAR

VAR
	ptIn 	: POINTER TO ST_FurnaceIn;
	ptOut 	: POINTER TO ST_FurnaceOut;
END_VAR
ptIn := ADR(stRefIO.stIn);
ptOut := ADR(stRefIO.stOut);

stIn REF= ptIn^;
stOut REF= ptOut^;
END_METHOD

METHOD SetupTempSensor
VAR_INPUT	
	nAnalogIn1		: INT;
	nValue1			: LREAL;

	nAnalogIn2		: INT;
	nValue2			: LREAL;
END_VAR
fSlope:= (nValue1 - nValue2) / (nAnalogIn1 - nAnalogIn2);
fInitial := nValue1 - (fSlope * nAnalogIn1);
END_METHOD

PROPERTY Temperature : LREAL
GET
Temperature := fTemperature;
END_GET
END_PROPERTY

END_FUNCTION_BLOCK

// ---- POUs/Components/AxisDriver/Utilities/F_TargetWindowReached.TcPOU
FUNCTION F_TargetWindowReached : BOOL
VAR_INPUT
	fCurrentPos: LREAL;
	fTargetPos: LREAL;
	fWindow: LREAL;
END_VAR


F_TargetWindowReached := fCurrentPos >= (fTargetPos - fWindow) AND fCurrentPos <= (fTargetPos + fWindow);

END_FUNCTION

// ---- POUs/Plant/ST020_OvenB/FB_St020_OvenB.TcPOU
FUNCTION_BLOCK FB_St020_OvenB EXTENDS FB_StationBase
VAR_INPUT
END_VAR
VAR	
	// IO ref
	stIO				: REFERENCE TO ST_St020_IO;
	
	// station components
	fbAxis 			: FB_AxisDriver;
	fbAxisCh1 		: FB_AxisDriver;
	fbAxisCh2 		: FB_AxisDriver;
	
	// actor UIs, access to: iStatus, fPosition, iVisibleState, ..
	fbAxisUi		: FB_Axis_Ui;
	fbAxisCh1Ui		: FB_Axis_Ui;
	fbAxisCh2Ui		: FB_Axis_Ui;
	
	fbHeatingPlate	: FB_FurnaceDriver;
	
	// instance var's
	bStationDeaktiv	: BOOL;
END_VAR
VAR PERSISTENT
	fPickupPos		: LREAL;
END_VAR

/// 
/// Station 020 function block - Oven B
///

{attribute 'monitoring' := 'call'}
PROPERTY PRIVATE HomeSpeed : LREAL
GET
HomeSpeed := stLocalSettings.stDynStationSettings[E_St020_Settings.eSt020_Settings_HomeSpeed].fValue;
END_GET
END_PROPERTY

{attribute 'monitoring' := 'call'}
PROPERTY PRIVATE JogSpeed : LREAL
GET
JogSpeed := stLocalSettings.stDynStationSettings[E_St020_Settings.eSt020_Settings_JogSpeed].fValue;
END_GET
END_PROPERTY

{attribute 'monitoring' := 'call'}
PROPERTY PRIVATE JogSpeedCh : LREAL
GET
JogSpeedCh := stLocalSettings.stDynStationSettings[E_St020_Settings.eSt020_Settings_JogSpeedCh].fValue;
END_GET
END_PROPERTY

METHOD PROTECTED M_CallObjects : BOOL
VAR
END_VAR
//Heating Plate
fbHeatingPlate.Run();

// axis + UI
fbAxis.TorqueLimit := 1000;
fbAxis(
	bEnable := SafetyOk AND NOT fbAxisUi.stAxisManager.bDisable,
	bEnablePos := stSt030IHandling.bEnableOvenAxis OR fbAxisUi.stAxisManager.bDisableSoftLimits,
	bEnableNeg := stSt030IHandling.bEnableOvenAxis OR fbAxisUi.stAxisManager.bDisableSoftLimits
);
fbAxisUi(
	bInHome := bInHome,
	fbAxis := fbAxis,
	fVelocity := JogSpeed,
	diSelectedObjectIndex := stHmiManualIn.diSelectedObjectIndex,
	stHMIControlIn := stHmiManualIn.stManualAxis,
	stHMIControlOut := stHmiManualOut.stManualAxis,
	bJogP := stHmi.stIn.stSt020.bJogUp,
	bJogN := stHmi.stIn.stSt020.bJogDown,
	bEnableManual := EnableManual);

// axis CH1 + UI
fbAxisCh1(
	bEnable := SafetyOk AND NOT fbAxisCh1Ui.stAxisManager.bDisable,
	bEnablePos := TRUE,
	bEnableNeg := TRUE,
);
fbAxisCh1Ui(
	bInHome := bInHome,
	fbAxis := fbAxisCh1,
	fVelocity := JogSpeedCh,
	diSelectedObjectIndex := stHmiManualIn.diSelectedObjectIndex,
	stHMIControlIn := stHmiManualIn.stManualAxis,
	stHMIControlOut := stHmiManualOut.stManualAxis,
	bJogP := stHmi.stIn.stSt020.bJogCh1Inside,
	bJogN := stHmi.stIn.stSt020.bJogCh1Ouside,
	bEnableManual := EnableManual);
	
// axis CH2 + UI
fbAxisCh2(
	bEnable := SafetyOk AND NOT fbAxisCh2Ui.stAxisManager.bDisable,
	bEnablePos := TRUE,
	bEnableNeg := TRUE,
);
fbAxisCh2Ui(
	bInHome := bInHome,
	fbAxis := fbAxisCh2,
	fVelocity := JogSpeedCh,
	diSelectedObjectIndex := stHmiManualIn.diSelectedObjectIndex,
	stHMIControlIn := stHmiManualIn.stManualAxis,
	stHMIControlOut := stHmiManualOut.stManualAxis,
	bJogP := stHmi.stIn.stSt020.bJogCh2Inside,
	bJogN := stHmi.stIn.stSt020.bJogCh2Ouside,
	bEnableManual := EnableManual);


// HMI : switch between jo modes
//IF stHmi.stIn.stSt020.bJog THEN
//	fbAxisUi.ManualMode :=  SEL(stHmi.stIn.stSt020.bSpeed, E_ManualMode.eManualMode_Jog01, E_ManualMode.eManualMode_Jog1);
//	fbAxisCh1Ui.ManualMode :=  SEL(stHmi.stIn.stSt020.bSpeed, E_ManualMode.eManualMode_Jog01, E_ManualMode.eManualMode_Jog1);
//	fbAxisCh2Ui.ManualMode :=  SEL(stHmi.stIn.stSt020.bSpeed, E_ManualMode.eManualMode_Jog01, E_ManualMode.eManualMode_Jog1);
//ELSE
//	fbAxisUi.ManualMode := E_ManualMode.eManualMode_Tippen;//	  SEL(stHmi.stIn.stSt020.bSpeed, E_ManualMode.eManualMode_TippSlow, E_ManualMode.eManualMode_TippFast);
//	fbAxisCh1Ui.ManualMode :=  E_ManualMode.eManualMode_Tippen;//		SEL(stHmi.stIn.stSt020.bSpeed, E_ManualMode.eManualMode_TippSlow, E_ManualMode.eManualMode_TippFast);
//	fbAxisCh2Ui.ManualMode :=  E_ManualMode.eManualMode_Tippen;//		SEL(stHmi.stIn.stSt020.bSpeed, E_ManualMode.eManualMode_TippSlow, E_ManualMode.eManualMode_TippFast);
//END_IF	
	
// run trolley logic
//Plant.stSt020IOvenB.Trolley.Update();
END_METHOD

METHOD INTERNAL M_DynManual : BOOL
VAR_INPUT
END_VAR
IF NOT bInitManual THEN
	bInitManual := TRUE;
	MEMSET(ADR(stHmiManualOut.stObjects), 0, SIZEOF(stHmiManualOut.stObjects)); // reset
	
	M_InitDynManualUi(fbAxisUi);
	M_InitDynManualUi(fbAxisCh1Ui);
	M_InitDynManualUi(fbAxisCh2Ui);
	
	fbAxisUi.M_TargetListClear();
	fbAxisUi.M_TargetListAddItem(F_CreateDynText("Home pos", 0), 15);
END_IF
END_METHOD

METHOD PROTECTED M_DynMonitoring : BOOL
VAR_INPUT
END_VAR
M_DynMonitoring := SUPER^.M_DynMonitoring();

// init
IF NOT bInitMonitoring THEN
	bInitMonitoring := TRUE;
	MEMSET(ADR(stLocalMonitoring), 0, SIZEOF(stLocalMonitoring)); // reset
	
	M_InitDynMonitoringItem(0, 								// monitoring index 
							"Achse Position", 				// name
							Name, 							// group (station name)
							E_DataType.eDataType_lreal, 	// data type							
							stTextListGlobal.stText_mm);	// unit	

	M_InitDynMonitoringItem(1, "Achse Geschwindigkeit", Name, E_DataType.eDataType_lreal, stTextListGlobal.stText_mms);
	M_InitDynMonitoringItem(2, "Achse Drehmoment", Name, E_DataType.eDataType_lreal, stTextListGlobal.stText_percent);
	
	M_InitDynMonitoringItem(4, "Achse CH1 Position", Name, E_DataType.eDataType_lreal, stTextListGlobal.stText_mm);
	M_InitDynMonitoringItem(5, "Achse CH1 Geschwindigkeit", Name, E_DataType.eDataType_lreal, stTextListGlobal.stText_mms);
	M_InitDynMonitoringItem(6, "Achse CH1 Drehmoment", Name, E_DataType.eDataType_lreal, stTextListGlobal.stText_percent);
	
	M_InitDynMonitoringItem(8, "Achse CH2 Position", Name, E_DataType.eDataType_lreal, stTextListGlobal.stText_mm);
	M_InitDynMonitoringItem(9, "Achse CH2 Geschwindigkeit", Name, E_DataType.eDataType_lreal, stTextListGlobal.stText_mms);
	M_InitDynMonitoringItem(10, "Achse CH2 Drehmoment", Name, E_DataType.eDataType_lreal, stTextListGlobal.stText_percent);
END_IF

// live value mapping 

// axis
stLocalMonitoring.astMonitoring[0].fValue := fbAxis.Position;
stLocalMonitoring.astMonitoring[1].fValue := fbAxis.Velocity;
stLocalMonitoring.astMonitoring[2].fValue := fbAxis.Torque;

// axis ch1
stLocalMonitoring.astMonitoring[4].fValue := fbAxisCh1.Position;
stLocalMonitoring.astMonitoring[5].fValue := fbAxisCh1.Velocity;
stLocalMonitoring.astMonitoring[6].fValue := fbAxisCh1.Torque;

// axis ch2
stLocalMonitoring.astMonitoring[8].fValue := fbAxisCh2.Position;
stLocalMonitoring.astMonitoring[9].fValue := fbAxisCh2.Velocity;
stLocalMonitoring.astMonitoring[10].fValue := fbAxisCh2.Torque;

// hmi value mapping
//HMI.stHmi.stOut.stSt020.Trolley := stSt020IOvenB.Trolley.stTrolley;
END_METHOD

METHOD INTERNAL M_DynSettings : BOOL
VAR
END_VAR
// init station settings
IF NOT bInitSettings THEN
	bInitSettings := TRUE;
	stLocalSettingsBackup := stLocalSettings; // backup
	MEMSET(ADR(stLocalSettings), 0, SIZEOF(stLocalSettings)); // reset
		
	Services.stSettings.stTrolley.CarrierConfig := Services.stSettings.stCarrier;
	stSt020IOvenB.Trolley.Config := Services.stSettings.stTrolley;
	stSt020IOvenB.Trolley.InitialStatus := eTcaWorkpieceStatus.laserProcessDone;
	stSt020IOvenB.Trolley.RequestStatus := eTcaWorkpieceStatus.castingProcessDone;
	stSt020IOvenB.Trolley.ApplyConfig();
	stSt020IOvenB.Trolley.FillWithInitialCarriers();
	
	M_InitDynSettingsItem(E_St020_Settings.eSt020_Settings_Station_Deaktiv,	// settings index
		TO_WSTRING(E_St020_Settings.eSt020_Settings_Station_Deaktiv),		// settings wsIndex
		Name,																// group
		stTextListGlobal.stText_DeactivateStation,							// name
		stTextListGlobal.stText_bool, E_DataType.eDataType_bool,			// unit & data type
		0, 1, 6);															// min, max & user level

	M_InitDynSettingsItem(E_St020_Settings.eSt020_Settings_Autohome,
		TO_WSTRING(E_St020_Settings.eSt020_Settings_Autohome),
		Name,
		stTextListGlobal.stText_AutoHome,
		stTextListGlobal.stText_bool, E_DataType.eDataType_bool,
		0, 1, 3);
		
	M_InitDynSettingsItem(E_St020_Settings.eSt020_Settings_HomeSpeed,
		TO_WSTRING(E_St020_Settings.eSt020_Settings_HomeSpeed),
		Name,
		F_CreateDynTextDefault("Homegeschwindigkeit Servoachse"),
		stTextListGlobal.stText_mms, E_DataType.eDataType_lreal,
		0, 50, 3);
		
	M_InitDynSettingsItem(E_St020_Settings.eSt020_Settings_JogSpeed,
		TO_WSTRING(E_St020_Settings.eSt020_Settings_JogSpeed),
		Name,
		F_CreateDynTextDefault("Tippgeschwindigkeit Servoachse"),
		stTextListGlobal.stText_mms, E_DataType.eDataType_lreal,
		0, 50, 3);
		
	M_InitDynSettingsItem(E_St020_Settings.eSt020_Settings_WorkSpeed,
		TO_WSTRING(E_St020_Settings.eSt020_Settings_WorkSpeed),
		Name,
		F_CreateDynTextDefault("Automatik-Geschwindigkeit Servoachse"),
		stTextListGlobal.stText_mms, E_DataType.eDataType_lreal,
		0, 500, 3);
		
	M_InitDynSettingsItem(E_St020_Settings.eSt020_Settings_JogSpeedCh,
		TO_WSTRING(E_St020_Settings.eSt020_Settings_JogSpeedCh),
		Name,
		F_CreateDynTextDefault("Tippgeschwindigkeit Servoachse CH"),
		stTextListGlobal.stText_mms, E_DataType.eDataType_lreal,
		0, 50, 3);
		
	M_InitDynSettingsItem(E_St020_Settings.eSt020_Settings_WorkSpeedCh,
		TO_WSTRING(E_St020_Settings.eSt020_Settings_WorkSpeedCh),
		Name,
		F_CreateDynTextDefault("Automatik-Geschwindigkeit Servoachse CH"),
		stTextListGlobal.stText_mms, E_DataType.eDataType_lreal,
		0, 500, 3);
		
	M_InitDynSettingsItem(E_St020_Settings.eSt020_Settings_AxisRefPos,
		TO_WSTRING(E_St020_Settings.eSt020_Settings_AxisRefPos),
		Name,
		F_CreateDynTextDefault("Referenzposition Achse Ofen"),
		stTextListGlobal.stText_m, E_DataType.eDataType_lreal,
		0, 3000, 6);
		
	M_InitDynSettingsItem(E_St020_Settings.eSt020_Settings_PosHome,
		TO_WSTRING(E_St020_Settings.eSt020_Settings_PosHome),
		Name,
		F_CreateDynTextDefault("Homeposition Servoachse"),
		stTextListGlobal.stText_mm, E_DataType.eDataType_lreal,
		0, 5000, 3);
		
	M_InitDynSettingsItem(E_St020_Settings.eSt020_Settings_PosWork,
		TO_WSTRING(E_St020_Settings.eSt020_Settings_PosWork),
		Name,
		F_CreateDynTextDefault("Mitnehmerposition unteres Segment"),
		stTextListGlobal.stText_mm, E_DataType.eDataType_lreal,
		0, 5000, 3);
		
	M_InitDynSettingsItem(E_St020_Settings.eSt020_Settings_PosHomeCh,
		TO_WSTRING(E_St020_Settings.eSt020_Settings_PosHomeCh),
		Name,
		F_CreateDynTextDefault("Homeposition Servoachse CH"),
		stTextListGlobal.stText_mm, E_DataType.eDataType_lreal,
		0, 500, 3);
		
	M_InitDynSettingsItem(E_St020_Settings.eSt020_Settings_PosWorkCh,
		TO_WSTRING(E_St020_Settings.eSt020_Settings_PosWorkCh),
		Name,
		F_CreateDynTextDefault("Arbeitsposition Servoachse CH"),
		stTextListGlobal.stText_mm, E_DataType.eDataType_lreal,
		0, 500, 3);
		
	M_InitDynSettingsItem(E_St020_Settings.eSt020_Settings_OvenFixPartHeight,
		TO_WSTRING(E_St020_Settings.eSt020_Settings_OvenFixPartHeight),
		Name,
		F_CreateDynTextDefault("Festteilhöhe"),
		stTextListGlobal.stText_mm, E_DataType.eDataType_lreal,
		0, 500, 3);
		
	M_InitDynSettingsItem(E_St020_Settings.eSt020_Settings_OvenSegmentHeight,
		TO_WSTRING(E_St020_Settings.eSt020_Settings_OvenSegmentHeight),
		Name,
		F_CreateDynTextDefault("Segmenthöhe"),
		stTextListGlobal.stText_mm, E_DataType.eDataType_lreal,
		0, 500, 3);				
	
	M_InitDynSettingsItem(E_St020_Settings.eSt020_Settings_OvenMiddlePointX,
		TO_WSTRING(E_St020_Settings.eSt020_Settings_OvenMiddlePointX),
		Name,
		F_CreateDynTextDefault("Mittelpunnkt in X-Richtung"),
		stTextListGlobal.stText_mm, E_DataType.eDataType_lreal,
		0, 500, 3);
		
	M_InitDynSettingsItem(E_St020_Settings.eSt020_Settings_OvenOffsetY,
		TO_WSTRING(E_St020_Settings.eSt020_Settings_OvenOffsetY),
		Name,
		F_CreateDynTextDefault("Y-Offset Ofen"),
		stTextListGlobal.stText_mm, E_DataType.eDataType_lreal,
		0, 500, 3);

	M_InitDynSettingsItem(E_St020_Settings.eSt020_Settings_OvenPickUpDepthZ,
		TO_WSTRING(E_St020_Settings.eSt020_Settings_OvenPickUpDepthZ),
		Name,
		F_CreateDynTextDefault("Oven Pick up Depth Z"),
		stTextListGlobal.stText_mm, E_DataType.eDataType_lreal,
		0, 5000, 3);

	M_InitDynSettingsItem(E_St020_Settings.eSt020_Settings_XPosRp1,	// Teach-Position, Ofen 2, RP 1
		TO_WSTRING(E_St020_Settings.eSt020_Settings_XPosRp1),
		Name,
		F_CreateDynTextDefault("Teach-Position, Ofen 2, RP 1 X"),
		stTextListGlobal.stText_mm, E_DataType.eDataType_lreal,
		0, 5000, 3);
	M_InitDynSettingsItem(E_St020_Settings.eSt020_Settings_YPosRp1,
		TO_WSTRING(E_St020_Settings.eSt020_Settings_YPosRp1),
		Name,
		F_CreateDynTextDefault("Teach-Position, Ofen 2, RP 1 Y"),
		stTextListGlobal.stText_mm, E_DataType.eDataType_lreal,
		0, 3000, 3);
	M_InitDynSettingsItem(E_St020_Settings.eSt020_Settings_ZPosRp1,
		TO_WSTRING(E_St020_Settings.eSt020_Settings_ZPosRp1),
		Name,
		F_CreateDynTextDefault("Teach-Position, Ofen 2, RP 1 Z"),
		stTextListGlobal.stText_mm, E_DataType.eDataType_lreal,
		0, 1000, 3);
		
	M_InitDynSettingsItem(E_St020_Settings.eSt020_Settings_XPosRp2,	// Teach-Position, Ofen 2, RP 2
		TO_WSTRING(E_St020_Settings.eSt020_Settings_XPosRp2),
		Name,
		F_CreateDynTextDefault("Teach-Position, Ofen 2, RP 2 X"),
		stTextListGlobal.stText_mm, E_DataType.eDataType_lreal,
		0, 5000, 3);
	M_InitDynSettingsItem(E_St020_Settings.eSt020_Settings_YPosRp2,
		TO_WSTRING(E_St020_Settings.eSt020_Settings_YPosRp2),
		Name,
		F_CreateDynTextDefault("Teach-Position, Ofen 2, RP 2 Y"),
		stTextListGlobal.stText_mm, E_DataType.eDataType_lreal,
		0, 3000, 3);
	M_InitDynSettingsItem(E_St020_Settings.eSt020_Settings_ZPosRp2,
		TO_WSTRING(E_St020_Settings.eSt020_Settings_ZPosRp2),
		Name,
		F_CreateDynTextDefault("Teach-Position, Ofen 2, RP 2 Z"),
		stTextListGlobal.stText_mm, E_DataType.eDataType_lreal,
		0, 1000, 3);
	

		
	// restore values
	F_RestoreSettingValues(stLocalSettings.stDynStationSettings, stLocalSettingsBackup.stDynStationSettings);
END_IF

// map current settings values
bStationDeaktiv := stLocalSettings.stDynStationSettings[E_St020_Settings.eSt020_Settings_Station_Deaktiv].bValue;
bAutoHome := stLocalSettings.stDynStationSettings[E_St020_Settings.eSt020_Settings_Autohome].bValue;
END_METHOD

METHOD PROTECTED M_Homing
VAR
	stHomPrm : ST_AxisHomingParameter;
END_VAR
// Homing sequence
CASE sqHome.Step OF
	
	0:	
		sqHome.Info.Set("Warte auf GRST Start");
		IF RunStep AND NOT sqHome.InHome AND bRunHoming THEN
			stSt020IOvenB.bResponseOpn := FALSE;
			bBusy := TRUE;
			sqAuto.Step := 0;
			sqHome.StartSequence()
				  .Step := 10;
		END_IF	

	10:
		sqHome.Info.Set("Grundstellungsfahrt aktiv");
		IF P_Safety.bMachineRequestStop THEN
			sqHome.Info.Set("Anforderung Stop aktiv");
		ELSIF NOT SafetyOk THEN
			sqHome.Info.Set("Sicherheit nicht ok");
			
		ELSIF NOT fbAxis.Operational THEN
			sqHome.Info.Set("Antrieb Ofen nicht bereit");
		ELSIF fbAxis.Moving THEN
			fbAxis.Halt();
			sqHome.Info.Set("Antrieb Ofen nicht gestoppt");
		ELSIF NOT stSt030IHandling.bEnableOvenAxis THEN
			sqHome.Info.Set("Warte auf Fahrfreigabe vom HG");
			
		ELSIF NOT fbAxisCh1.Operational THEN
			sqHome.Info.Set("Antrieb Ofen CH1 nicht bereit");
		ELSIF fbAxisCh1.Moving THEN
			fbAxisCh1.Halt();
			sqHome.Info.Set("Antrieb Ofen CH1 nicht gestoppt");
			
		ELSIF NOT fbAxisCh2.Operational THEN
			sqHome.Info.Set("Antrieb Ofen CH2 nicht bereit");
		ELSIF fbAxisCh2.Moving THEN
			fbAxisCh2.Halt();
			sqHome.Info.Set("Antrieb Ofen CH2 nicht gestoppt");

		ELSIF bRunHoming THEN
			sqHome.Step := 15;
		END_IF
		
	15:	sqHome.Info.Set("Prüfe Status");
		IF F_TargetWindowReached(fbAxisCh1.Position, PosHomeCh, chAxisPosTol) AND 
		   F_TargetWindowReached(fbAxisCh2.Position, PosHomeCh, chAxisPosTol) THEN
			sqHome.SetStep(20);
		ELSIF fbAxis.Homed THEN
			sqHome.SetStep(16); // close segment
		ELSE
			StationError.ArgSbAppendRaise('Segmenttor manuell schließen!');
		END_IF
		
	16: sqHome.Info.Set("Start Achse zu Arbeitspos.");
		fbAxis.MoveAbsExVel(fPickupPos, WorkSpeed);
		sqHome.Step := 17;
		
	17: sqHome.Info.Set("Warte auf Achse in Arbeitspos");
		IF fbAxis.TargetReached() THEN
			sqHome.SetStep(20); // ch axis back
		END_IF
	
	20:
		sqHome.Info.Set("Grundstellungsfahrt aktiv Achse CH1 auf Homepos.");
		fbAxisCh1.MoveAbsExVel(PosHomeCh, WorkSpeedCh);
		sqHome.Step := 25;
		
	25:
		sqHome.Info.Set("Warte auf Achse CH1 in Homeposition");
		IF fbAxisCh1.TargetWindowReached(chAxisPosTol) THEN
			sqHome.Step := 30;
		END_IF
		
	30:
		sqHome.Info.Set("Grundstellungsfahrt aktiv Achse CH2 auf Homepos.");
		fbAxisCh2.MoveAbsExVel(PosHomeCh, WorkSpeedCh);
		sqHome.Step := 35;
		
	35:
		sqHome.Info.Set("Warte auf Achse CH2 in Homeposition");
		IF fbAxisCh2.TargetWindowReached(chAxisPosTol) THEN
			sqHome.Step := 40;
		END_IF
	
	40:
		sqHome.Info.Set("Prüfe Achskalibrierung");
		IF fbAxis.Homed THEN
			sqHome.Step := 50;
		ELSE
			sqHome.Step := 42;
		END_IF
		
	42:
		sqHome.Info.Set("Starte Achskalibrierung");
		IF RunStep THEN
			stHomPrm.fPosition := OvenRefPos;
			stHomPrm.stOptions.SearchDirection := MC_Direction.MC_Negative_Direction;
			stHomPrm.stOptions.SyncDirection := MC_Direction.MC_Positive_Direction;
			stHomPrm.stOptions.SearchVelocity := 8;
			stHomPrm.stOptions.SyncVelocity := 4;
			fbAxis.HomeEx(stHomPrm);
			sqHome.Step := 44;
		END_IF
		
	44:
		sqHome.Info.Set("Warte auf Achskalibrierung fertig");
		fbAxis.bCalibrationCam := stIO.stIn.bRefpos;
		IF fbAxis.Homed THEN
			sqHome.Step := 50;
		END_IF
		
	50:
		sqHome.Info.Set("Grundstellungsfahrt aktiv Achse auf Homepos.");
		fbAxis.MoveAbsExVel(PosHome, HomeSpeed);
		sqHome.Step := 60;
		
	60:
		sqHome.Info.Set("Warte auf Achse in Homeposition");
		IF fbAxis.TargetReached() THEN
			sqHome.Step := 100;
		END_IF
		
	100:
		sqHome.Info.Set("Grundstellungsfahrt aktiv");
		sqHome.Step := 1000;

	//	homing done			
	1000:
		sqHome.Info.Set("Grundstellung erreicht");
		IF sqHome.StepTime > T#1S THEN		
			bBusy:=FALSE;
			sqHome.InHome := TRUE;
			bStopped := TRUE;
			bRunHoming := FALSE;
			sqAuto.Step := 0;
			sqHome.StopSequence()
				  .Step := 0;
		END_IF
END_CASE
END_METHOD

METHOD PUBLIC M_Init : IStation
VAR_INPUT
END_VAR
VAR
	Ist : IStation;
END_VAR
// set up station
StationNb := 20;
Station := E_Station.eStation_ST020_OvenB; // ID & name 1st!
Name := F_CreateDynTextEx(1, "ST020_OvenB", "ST020 Ofen B");

Ist := SUPER^.M_Init()
			 .InitEvents(TC_Events.ST020EventClass.InfoEvent,
	  		       		 TC_Events.ST020EventClass.WarningEvent,
	  				  	 TC_Events.ST020EventClass.ErrorEvent);

// set up default IO references
M_SetReferences(IO.st020_OvenB_IO);

// init components

// Axis
fbAxisUi.stBmk := F_CreateDynTextDefault("BMK=A03.ST20.M01-");
fbAxisUi.stUnit := F_CreateDynTextDefault("mm");
fbAxisUi.stAxisManager.bEnablePosSet := TRUE;
fbAxisUi.stAxisManager.bSetCalibrationVisible := TRUE;
fbAxisUi.stAxisManager.bResetCalibrationVisible := TRUE;
fbAxis.AxisId := TO_INT(E_Axis.eAxis_OvenB);
fbAxis.Active := TRUE;
fbAxis.Name := F_CreateDynTextEx(1, "ServoOvenB", "Servoachse Ofen B");
fbAxis.AxisType := E_AxisType.AX5xxx;
//fbAxis.DefaultParameter := F_GetDefaultMotionParameter(eMainState_setup);
fbAxis.SetAxisReference(NcIO.stAxis_ST020_OvenB, NcIO.stAxis_ST020_OvenB_IO.stIn, NCIO.stAxis_ST020_OvenB_IO.stOut);

// Axis CH1
fbAxisCh1Ui.stBmk := F_CreateDynTextDefault("BMK=A03.ST20.M02-");
fbAxisCh1Ui.stUnit := F_CreateDynTextDefault("mm");
fbAxisCh1Ui.stAxisManager.bEnablePosSet := TRUE;
fbAxisCh1.AxisId := TO_INT(E_Axis.eAxis_OvenB_CH1);
fbAxisCh1.Active := TRUE;
fbAxisCh1.Name := F_CreateDynTextEx(1, "ServoOvenBCh1", "Servoachse Ofen B CH1");
fbAxisCh1.AxisType := E_AxisType.AX5xxx;
//fbAxisCh1.DefaultParameter := F_GetDefaultMotionParameter(eMainState_setup);
fbAxisCh1.SetAxisReference(NcIO.stAxis_ST020_OvenBCh1, NcIO.stAxis_ST020_OvenBCh1_IO.stIn, NCIO.stAxis_ST020_OvenBCh1_IO.stOut);

// Axis CH2
fbAxisCh2Ui.stBmk := F_CreateDynTextDefault("BMK=A03.ST20.M03-");
fbAxisCh2Ui.stUnit := F_CreateDynTextDefault("mm");
fbAxisCh2Ui.stAxisManager.bEnablePosSet := TRUE;
fbAxisCh2.AxisId := TO_INT(E_Axis.eAxis_OvenB_CH2);
fbAxisCh2.Active := TRUE;
fbAxisCh2.Name := F_CreateDynTextEx(1, "ServoOvenBCh2", "Servoachse Ofen B CH2");
fbAxisCh2.AxisType := E_AxisType.AX5xxx;
//fbAxisCh2.DefaultParameter := F_GetDefaultMotionParameter(eMainState_setup);
fbAxisCh2.SetAxisReference(NcIO.stAxis_ST020_OvenBCh2, NcIO.stAxis_ST020_OvenBCh2_IO.stIn, NCIO.stAxis_ST020_OvenBCh2_IO.stOut);

// register station in it's module
eParent := fbModul001.M_RegisterStation(Ist);

bInitSettings	:= FALSE;
bInitMonitoring := FALSE;
bInitManual  	:= FALSE;

//aSClearText[EN] := 'Station init done.';
M_Init := Ist;
END_METHOD

METHOD PROTECTED M_Manual
VAR
	fbTR : REFERENCE TO TcaTrolley;
END_VAR

// station must be stopped!			manual mode
IF RunCycle OR NOT bStopped THEN //(OpMode <> E_OpMode.eOpMode_manual) THEN
	RETURN;
END_IF

stSt020IOvenB.Trolley.ServiceMode();

//IF stHmiInOut.stSt020.Command = E_HMI_TR_CMD.eHmiTrCmd_none AND_THEN 
//   stHmiInOut.stSt020.PlCmd.Command <> E_HMI_PL_CMD.eHmiPlCmd_none THEN
//	stHmiInOut.stSt020.Command := E_HMI_TR_CMD.eHmiTrCmd_performPlCmd;
//END_IF
//
//IF stHmiInOut.stSt020.Command = E_HMI_TR_CMD.eHmiTrCmd_performPlCmd THEN
//	RETURN;
//END_IF
//
//stSt020IOvenB.Trolley.PerformHmiCmd(stHmiInOut.stSt020);
END_METHOD

METHOD PROTECTED M_OpModeChanged : BOOL
VAR_INPUT
END_VAR
(*bBusy := FALSE;

IF (eOpMode <> eOpMode_step AND eOpMode <> eOpMode_auto) THEN
	sqAuto.Set(0);
END_IF

fbAxis.Stop();
fbAxisCh1.Stop();
fbAxisCh2.Stop();*)
END_METHOD

METHOD PUBLIC M_Run : BOOL
VAR_INPUT
END_VAR
// check refs valid
IF NOT __ISVALIDREF(stIO) THEN
	RETURN;
END_IF

M_RUN := SUPER^.M_Run();

M_DynSettings();
M_DynManual();
M_DynMonitoring();
END_METHOD

METHOD PROTECTED M_Sequence
VAR
	fTmp : LREAL;
END_VAR
// signal mapping (e.g.: enable)
stSt020IOvenB.bEnableSequence := (sqAuto.Step = 100 AND fbAxis.Operational AND fbAxisCh1.Operational AND fbAxisCh2.Operational) OR
									bStationDeaktiv;

// automatic sequence
CASE sqAuto.Step OF
	
	0:	sqAuto.Info.Set("Warte auf Auto Start");
		IF RunCycle AND RunStep THEN
			//sqAuto.Info.Set("Warte auf GRST");
			//IF sqAuto.InHome AND bInHome THEN
				sqAuto.InHome := FALSE;
				sqAuto.Step := 10;
			//ELSE
			//	StationError.ArgSbAppendWsRaise(stTextlistGlobal.stText_station_not_in_hp);
			//END_IF
		END_IF
		
	10:	sqAuto.Info.Set("Prüfe Startbedingungen");
		IF NOT (fbAxis.Operational AND fbAxis.Homed) THEN
			StationError.ArgSbAppendRaise('Achse nicht bereit');
		ELSIF NOT fbAxisCh1.Operational THEN
			StationError.ArgSbAppendRaise('Achse CH1 nicht bereit');
		ELSIF NOT fbAxisCh2.Operational THEN
			StationError.ArgSbAppendRaise('Achse CH2 nicht bereit');
		ELSE
			CycleStart();
			//stSt020IOvenB.bStorageEnd := FALSE;
			sqAuto.Step := 15;
		END_IF
		
	15:	sqAuto.Info.Set("Prüfe Status");
		IF F_TargetWindowReached(fbAxisCh1.Position, PosHomeCh, chAxisPosTol) AND 
		   F_TargetWindowReached(fbAxisCh2.Position, PosHomeCh, chAxisPosTol) THEN
			sqAuto.SetStep(20);
		ELSE
			sqAuto.SetStep(160); // close segment
		END_IF
		
	20:	sqAuto.Info.Set("Start Achse CH1 auf Homepos.");
		fbAxisCh1.MoveAbsExVel(PosHomeCh, WorkSpeedCh);
		fbAxisCh2.MoveAbsExVel(PosHomeCh, WorkSpeedCh);
		sqAuto.Step := 30;
		
	30:	sqAuto.Info.Set("Warte Achse CH1 in Homeposition");
		IF NOT fbAxisCh1.TargetWindowReached(chAxisPosTol) THEN RETURN; END_IF
		sqAuto.Info.Set("Warte Achse CH2 in Homeposition");
		IF NOT fbAxisCh2.TargetWindowReached(chAxisPosTol) THEN RETURN; END_IF
		sqAuto.SetStep(100);

	// work
	100: sqAuto.Info.Set("Automatik, warte auf Anforderung vom HG");
		IF stSt030IHandling.bReqestOvenB_ChkIndex THEN
			sqAuto.Info.Append(", Index-Check");
			stSt020IOvenB.iConfirmPosition := stSt030IHandling.ActiveCommand.Position;
			stSt020IOvenB.bResponseIsEmptySlot := stSt020IOvenB.Trolley.IsEmptySlotAt(stSt020IOvenB.iConfirmPosition);
			stSt020IOvenB.bResponseChkIndex := TRUE;
			IF stSt030IHandling.bReqestOvenB THEN sqAuto.SetStep(110); END_IF
		END_IF
	
		IF RunCycle THEN RETURN; END_IF
		sqAuto.Info.Set("Stop - warte auf Ablauf gestoppt");
		sqAuto.Step := 900;
		
	110: sqAuto.Info.Set("Start Achse zu Arbeitspos.");
		fPickupPos := PosWork;
		fbAxis.MoveAbsExVel(fPickupPos, WorkSpeed);
		sqAuto.Step := 115;
		
	115: sqAuto.Info.Set("Warte auf Achse in Arbeitspos");
		IF fbAxis.TargetReached() THEN
			sqAuto.SetStep(120);
		END_IF
		
	120: sqAuto.Info.Set("Start Achse CH1 zu Arbeitspos.");
		fbAxisCh1.MoveAbsExVel(PosWorkCh, WorkSpeedCh);
		fbAxisCh2.MoveAbsExVel(PosWorkCh, WorkSpeedCh);
		sqAuto.Step := 125;
		
	125: sqAuto.Info.Set("Warte Achse CH1 in Arbeitspos");
		IF fbAxisCh1.TargetWindowReached(chAxisPosTol) THEN
			sqAuto.SetStep(130);
		END_IF
		
	130: sqAuto.Info.Set("Start Achse CH2 zu Arbeitspos.");
		fbAxisCh2.MoveAbsExVel(PosWorkCh, WorkSpeedCh);
		sqAuto.Step := 135;
		
	135: sqAuto.Info.Set("Warte Achse CH2 in Arbeitspos");
		IF fbAxisCh2.TargetWindowReached(chAxisPosTol) THEN
			sqAuto.SetStep(140);
		END_IF
		
	140: sqAuto.Info.Set("Start Achse zu Arbeitspos. offen");
		fTmp := (PosWorkOpn - PosWork);
		IF fTmp > 540 THEN
			sqAuto.Info.Set("Max. Öffnungsweg überschritten: ")
					   .AppendAny(fTmp);
			
			StationError.ArgSbAppendS(sqAuto.Info.ToString())
						.Raise();
			RETURN;
		END_IF
		fbAxis.MoveAbsExVel(PosWorkOpn, WorkSpeed);
		sqAuto.Step := 145;
		
	145: sqAuto.Info.Set("Warte auf Achse in Arbeitspos. offen");
		IF fbAxis.TargetReached() THEN
			sqAuto.Step := 150;
		END_IF
		
	150: sqAuto.Info.Set("Segment offen, warte auf Anforderung vom HG");
		stSt020IOvenB.bResponseOpn := TRUE;
		IF NOT stSt030IHandling.bReqestOvenB THEN
			stSt020IOvenB.bResponseOpn := FALSE;
			sqAuto.SetStep(160);
		END_IF
		
	160: sqAuto.Info.Set("Start Achse zu Arbeitspos.");
		fbAxis.MoveAbsExVel(fPickupPos, WorkSpeed);
		sqAuto.Step := 165;
		
	165: sqAuto.Info.Set("Warte auf Achse in Arbeitspos");
		IF fbAxis.TargetReached() THEN
			sqAuto.SetStep(170);
		END_IF
		
	170: sqAuto.Info.Set("Start Achse CH1 auf Homepos.");
		fbAxisCh1.MoveAbsExVel(PosHomeCh, WorkSpeedCh);
		fbAxisCh2.MoveAbsExVel(PosHomeCh, WorkSpeedCh);
		sqAuto.Step := 175;
		
	175:	sqAuto.Info.Set("Warte Achse CH1 in Homeposition");
		IF NOT fbAxisCh1.TargetWindowReached(chAxisPosTol) THEN RETURN; END_IF
		sqAuto.Info.Set("Warte Achse CH2 in Homeposition");
		IF NOT fbAxisCh2.TargetWindowReached(chAxisPosTol) THEN RETURN; END_IF
		sqAuto.SetStep(900);
		
	// rdy	
	900: sqAuto.Info.Set("Zyklus beendet");
		CycleEnd();
		sqAuto.Step := 0; // ch axis back, loop

	// error
	1000: sqAuto.Info.Set("Error");
		bStopped := TRUE;
		sqAuto.InHome := FALSE;
		bRunHoming := FALSE;

END_CASE
END_METHOD

METHOD INTERNAL M_SetReferences : BOOL
VAR_IN_OUT
	stIoRef : ST_St020_IO;
END_VAR
stIO REF= stIoRef;
M_SetReferences := TRUE;

fbHeatingPlate.SetReferences(stIoRef.stHeatingPlateIO);
fbHeatingPlate.LoadCtrlParam();
fbHeatingPlate.CtrlParameter.tPWMCycleTime := T#5S;
fbHeatingPlate.PIDParameter.KpHeat := 41.3793103448273;
fbHeatingPlate.PIDParameter.TnHeat := T#29S;
fbHeatingPlate.PIDParameter.TvHeat := T#6S90MS; 
fbHeatingPlate.PIDParameter.TdHeat := T#1S523MS; 
fbHeatingPlate.SetupTempSensor(0,0,100,10);
END_METHOD

METHOD PROTECTED M_Supervision : BOOL
VAR
END_VAR
// chk stopped
IF NOT bRunCycle OR P_Safety.bMachineRequestStop THEN
	IF P_Safety.bMachineRequestStop THEN
		fbAxis.Stop();
	END_IF
	IF sqAuto.StepTime > T#20S THEN
		bStopped := TRUE;
	END_IF
END_IF

// chk requested index
IF stSt030IHandling.bReqestOvenB_ChkIndex THEN
	;// --> confirm chk implemented in M_Sequence, step 100
	//stSt020IOvenB.iConfirmOpnIdxX := stSt030IHandling.ActiveCommand.IndexX;
	//stSt020IOvenB.iConfirmOpnIdxY := stSt030IHandling.ActiveCommand.IndexY;
	//stSt020IOvenB.bResponseIsEmptySlot := stSt020IOvenB.Trolley.IsEmptySlotAt(stSt020IOvenB.iConfirmOpnIdxX, stSt020IOvenB.iConfirmOpnIdxY);
	//stSt020IOvenB.bResponseChkIndex := TRUE;
ELSE
	stSt020IOvenB.iConfirmPosition := -1;
	stSt020IOvenB.bResponseIsEmptySlot := FALSE;
	stSt020IOvenB.bResponseChkIndex := FALSE;
END_IF

// axis
IF fbAxis.bError THEN
	ReactToComponentError(fbAxisUi, E_EventReaction.Stop);

// ch1
ELSIF fbAxisCh1.bError THEN
	ReactToComponentError(fbAxisCh1Ui, E_EventReaction.Stop);
	
// ch2
ELSIF fbAxisCh2.bError THEN
	ReactToComponentError(fbAxisCh2Ui, E_EventReaction.Stop);
	
END_IF
END_METHOD

{attribute 'monitoring' := 'call'}
PROPERTY PRIVATE OvenFixPartHeight : LREAL
GET
OvenFixPartHeight := stLocalSettings.stDynStationSettings[E_St020_Settings.eSt020_Settings_OvenFixPartHeight].fValue;
END_GET
END_PROPERTY

{attribute 'monitoring' := 'call'}
PROPERTY INTERNAL OvenMiddlePointX : LREAL
GET
OvenMiddlePointX := stLocalSettings.stDynStationSettings[E_St020_Settings.eSt020_Settings_OvenMiddlePointX].fValue;
END_GET
END_PROPERTY

{attribute 'monitoring' := 'call'}
PROPERTY INTERNAL OvenOffsetY : LREAL
GET
OvenOffsetY := stLocalSettings.stDynStationSettings[E_St020_Settings.eSt020_Settings_OvenOffsetY].fValue;
END_GET
END_PROPERTY

{attribute 'monitoring' := 'call'}
PROPERTY INTERNAL OvenPickUpDepthZ : LREAL
GET
OvenPickUpDepthZ := stLocalSettings.stDynStationSettings[E_St020_Settings.eSt020_Settings_OvenPickUpDepthZ].fValue;
END_GET
END_PROPERTY

{attribute 'monitoring' := 'call'}
PROPERTY INTERNAL OvenRefPos : LREAL
GET
OvenRefPos := stLocalSettings.stDynStationSettings[E_St020_Settings.eSt020_Settings_AxisRefPos].fValue;
END_GET
END_PROPERTY

{attribute 'monitoring' := 'call'}
PROPERTY PRIVATE OvenSegmentHeight : LREAL
GET
OvenSegmentHeight := stLocalSettings.stDynStationSettings[E_St020_Settings.eSt020_Settings_OvenSegmentHeight].fValue;
END_GET
END_PROPERTY

{attribute 'monitoring' := 'call'}
PROPERTY INTERNAL PosHome : LREAL
GET
PosHome := stLocalSettings.stDynStationSettings[E_St020_Settings.eSt020_Settings_PosHome].fValue;
END_GET
END_PROPERTY

{attribute 'monitoring' := 'call'}
PROPERTY INTERNAL PosHomeCh : LREAL
GET
PosHomeCh := stLocalSettings.stDynStationSettings[E_St020_Settings.eSt020_Settings_PosHomeCh].fValue;
END_GET
END_PROPERTY

{attribute 'monitoring' := 'call'}
PROPERTY INTERNAL PosWork : LREAL
GET
PosWork := stLocalSettings.stDynStationSettings[E_St020_Settings.eSt020_Settings_PosWork].fValue + // 1. Mitnehmerpos.
	  (OvenSegmentHeight * 
		TRUNC(((P_Plant.TrolleyRackDivision * stSt020IOvenB.iConfirmPosition) + (P_Plant.TrolleyRackOriginX - OvenFixPartHeight - 50))/OvenSegmentHeight));
END_GET
END_PROPERTY

{attribute 'monitoring' := 'call'}
PROPERTY INTERNAL PosWorkCh : LREAL
GET
PosWorkCh := stLocalSettings.stDynStationSettings[E_St020_Settings.eSt020_Settings_PosWorkCh].fValue;
END_GET
END_PROPERTY

{attribute 'monitoring' := 'call'}
PROPERTY INTERNAL PosWorkOpn : LREAL
GET
VAR
	_pos : ST_Coordinate;
END_VAR
_pos := stSt020IOvenB.Trolley.GetCoordinateAt(stSt020IOvenB.iConfirmPosition) ;

PosWorkOpn := PosWork + 
			  LMOD(_pos.fY - OvenFixPartHeight - 50, OvenSegmentHeight) + 					
			  50 + // -50 => height axis z
			  P_Plant.TrolleyRackDivision; // ( + TrolleyDevisionY --> safety distance)


//			  LMOD(((P_Plant.TrolleyDevisionY * stSt020IOvenB.iConfirmOpnIdxY) + (P_Plant.TrolleyFirstPosY - OvenFixPartHeight - 50)), 
//					P_Plant.OvenSegmHeight) + 
//					50 + // -50 => height axis z
//			  P_Plant.TrolleyDevisionY; // ( + TrolleyDevisionY --> safety distance)
END_GET
END_PROPERTY

/// Reset station logic
{attribute 'object_name' := 'Reset'}
METHOD Reset
VAR
END_VAR
// base logic run
SUPER^.Reset();

// reset objects
//diContinuesNok := 0;

IF fbAxis.bError OR NOT RunCycle THEN
	fbAxis.Reset();
END_IF
IF fbAxisCh1.bError OR NOT RunCycle THEN
	fbAxisCh1.Reset();
END_IF
IF fbAxisCh2.bError OR NOT RunCycle THEN
	fbAxisCh2.Reset();
END_IF
END_METHOD

{attribute 'monitoring' := 'call'}
PROPERTY PRIVATE WorkSpeed : LREAL
GET
WorkSpeed := stLocalSettings.stDynStationSettings[E_St020_Settings.eSt020_Settings_WorkSpeed].fValue;
END_GET
END_PROPERTY

{attribute 'monitoring' := 'call'}
PROPERTY PRIVATE WorkSpeedCh : LREAL
GET
WorkSpeedCh := stLocalSettings.stDynStationSettings[E_St020_Settings.eSt020_Settings_WorkSpeedCh].fValue;
END_GET
END_PROPERTY

END_FUNCTION_BLOCK

// ---- POUs/Items/TcaTrolley/TcaTrolley.TcPOU
FUNCTION_BLOCK TcaTrolley //EXTENDS TcoCore.TcoComponent
VAR CONSTANT
	MAX_CARRIERPLACES : INT := 39;
END_VAR

VAR PERSISTENT
	_data : TcaTrolleyData;
	_config : TcaTrolleyConfig;
	_service : TcaTrolleyService;
END_VAR

VAR	
	_CarriersCoordinate : ARRAY[0..TcaCarrier.MAX_WORKPIECEPLACES] OF ST_Coordinate;
	_TemplateCarrier : TcaCarrier;//(THIS^);
END_VAR

METHOD ApplyConfig
VAR
	_i : INT;
	_Coordinate 		: ST_Coordinate;	
	_CarrierPerSide		: INT;
END_VAR
MEMSET(ADR(_CarriersCoordinate),0,SIZEOF(_CarriersCoordinate));
MEMSET(ADR(_data.CarriersEnabled),0,SIZEOF(_data.CarriersEnabled));

_CarrierPerSide := _config.NumberOfCarriers/2;

FOR _i:=0 TO _config.NumberOfCarriers-1 DO
 	_Coordinate.fY  := _config.RackOrigin.fY +_config.CarrierDistance*(_i MOD(_CarrierPerSide));
 	_Coordinate.fX  := _config.RackOrigin.fX +_config.RackDivision/2*SEL(_i >= _CarrierPerSide, -1,  1);
	_CarriersCoordinate[_i] := _Coordinate;
	_data.CarriersEnabled[_i] := TRUE;
	_data.CarriersData[_i].Enabled := TRUE;
END_FOR

_TemplateCarrier.Config := _config.CarrierConfig;
_TemplateCarrier.ApplyConfig();
END_METHOD

PROPERTY Config : REFERENCE TO TcaTrolleyConfig
GET
Config REF= _config;
END_GET
SET
_config := Config;
END_SET
END_PROPERTY

PROPERTY Data : REFERENCE TO TcaTrolleyData
GET
Data REF= _data;
END_GET
SET
_data := Data;
END_SET
END_PROPERTY

{attribute 'TcRpcEnable'}
METHOD DisableCarriers
VAR
	_i :INT;
END_VAR
//MEMSET(ADR(_data.CarriersData),0,SIZEOF(_data.CarriersData));
FOR _i:=0 TO _config.NumberOfCarriers-1 DO
	//_data.CarriersEnabled[_i]:= FALSE;
	_data.CarriersData[_i].Enabled := FALSE;
END_FOR

//FOR _config.NumberOfCarriers:=0 TO MAX_CARRIERPLACES DO
//	_data.CarriersData[_i].Enabled := FALSE;
//END_FOR
END_METHOD

{attribute 'monitoring' := 'call'}
PROPERTY PUBLIC EmptySlot : INT
GET
VAR
	_i : INT;
END_VAR
EmptySlot:= -1;
	
FOR _i:= 0 TO MAX_CARRIERPLACES DO
	
	IF  _data.CarriersData[_i].Enabled THEN
		EmptySlot:= _i;
		RETURN;
	END_IF	

END_FOR
END_GET
END_PROPERTY

{attribute 'TcRpcEnable'}
METHOD EnableCarriers
VAR
	_i :INT;
END_VAR
//MEMSET(ADR(_data.CarriersData),0,SIZEOF(_data.CarriersData));
FOR _i:=0 TO _config.NumberOfCarriers-1 DO
	//_data.CarriersEnabled[_i]:= TRUE;
	_data.CarriersData[_i].Enabled := TRUE;
END_FOR

//FOR _config.NumberOfCarriers:=0 TO MAX_CARRIERPLACES DO
//	_data.CarriersData[_i].Enabled := FALSE;
//END_FOR
END_METHOD

{attribute 'TcRpcEnable'}
METHOD FillWithEmptyCarriers
VAR
	_i :INT;
END_VAR
_TemplateCarrier.Config := _config.CarrierConfig;
_TemplateCarrier.EmptyCarrier();

MEMSET(ADR(_data.CarriersData),0,SIZEOF(_data.CarriersData));
FOR _i:=0 TO _config.NumberOfCarriers-1 DO
	//_data.CarriersEnabled[_i]:= TRUE;
	_data.CarriersData[_i] := _TemplateCarrier.Data;
	_data.CarriersData[_i].Enabled := TRUE;
END_FOR

//FOR _config.NumberOfCarriers:=0 TO MAX_CARRIERPLACES DO
//	_data.CarriersData[_i].Enabled := FALSE;
//END_FOR
END_METHOD

{attribute 'TcRpcEnable'}
METHOD FIllWithFinishedCarriers
VAR
	_i :INT;
END_VAR
_TemplateCarrier.Config := _config.CarrierConfig;
_TemplateCarrier.FinishCarrier();

MEMSET(ADR(_data.CarriersData),0,SIZEOF(_data.CarriersData));
FOR _i:=0 TO _config.NumberOfCarriers-1 DO
	//_data.CarriersEnabled[_i]:= TRUE;
	_data.CarriersData[_i] := _TemplateCarrier.Data;
	_data.CarriersData[_i].Enabled := TRUE;
END_FOR

//FOR _config.NumberOfCarriers:=0 TO MAX_CARRIERPLACES DO
//	_data.CarriersData[_i].Enabled := FALSE;
//END_FOR
END_METHOD

{attribute 'TcRpcEnable'}
METHOD FillWithInitialCarriers 
VAR
	_i :INT;
END_VAR
_TemplateCarrier.Config := _config.CarrierConfig;
_TemplateCarrier.InitialCarrier();

MEMSET(ADR(_data.CarriersData),0,SIZEOF(_data.CarriersData));
FOR _i:=0 TO _config.NumberOfCarriers-1 DO
	//_data.CarriersEnabled[_i]:= TRUE;
	_data.CarriersData[_i] := _TemplateCarrier.Data;
	_data.CarriersData[_i].Enabled := TRUE;
END_FOR

//FOR _config.NumberOfCarriers:=0 TO MAX_CARRIERPLACES DO
//	_data.CarriersData[_i].Enabled := FALSE;
//END_FOR
END_METHOD

METHOD PUBLIC GetCarrierAt : TcaCarrierData
VAR_INPUT
	Position : INT;
END_VAR
IF Position < 0 OR Position > MAX_CARRIERPLACES OR NOT _data.CarriersEnabled[Position] THEN
   RETURN;
END_IF

GetCarrierAt := _data.CarriersData[Position];
END_METHOD

METHOD PUBLIC GetCarrierRefAt : Reference TO TcaCarrierData
VAR_INPUT
	Position : INT;
END_VAR
IF Position < 0 OR Position > MAX_CARRIERPLACES OR NOT _data.CarriersEnabled[Position] THEN
   RETURN;
END_IF

GetCarrierRefAt REF= _data.CarriersData[Position];
END_METHOD

METHOD GetCoordinateAt : ST_Coordinate
VAR_INPUT
	Position : INT;
END_VAR
IF Position < 0 OR Position > MAX_CARRIERPLACES OR NOT _data.CarriersEnabled[Position] THEN
   RETURN;
END_IF

GetCoordinateAt := _CarriersCoordinate[Position];
END_METHOD

{attribute 'monitoring' := 'call'}
PROPERTY PUBLIC HasCarrierWithEmptyWorkpieceplace : BOOL
GET
VAR
	_i : INT;
END_VAR
HasCarrierWithEmptyWorkpieceplace:= FALSE;
	
FOR _i:= 0 TO MAX_CARRIERPLACES DO

	THIS^._TemplateCarrier.Data := _data.CarriersData[_i];
	
	IF _TemplateCarrier.HasEmptyWorkpieceplaces THEN
		HasCarrierWithEmptyWorkpieceplace:= TRUE;
		RETURN;
	END_IF

END_FOR
END_GET
END_PROPERTY

{attribute 'monitoring' := 'call'}
PROPERTY PUBLIC HasCarrierWithInitialWorkpiece : BOOL
GET
VAR
	_i : INT;
END_VAR
HasCarrierWithInitialWorkpiece:= FALSE;
	
FOR _i:= 0 TO MAX_CARRIERPLACES DO

	THIS^._TemplateCarrier.Data := _data.CarriersData[_i];
	
	IF _TemplateCarrier.HasWorkpiecesWithInitialStatus THEN
		HasCarrierWithInitialWorkpiece:= TRUE;
		RETURN;
	END_IF

END_FOR
END_GET
END_PROPERTY

{attribute 'monitoring' := 'call'}
PROPERTY PUBLIC HasCarrierWithRequestWorkpiece : BOOL
GET
VAR
	_i : INT;
END_VAR
HasCarrierWithRequestWorkpiece:= FALSE;
	
FOR _i:= 0 TO MAX_CARRIERPLACES DO

	THIS^._TemplateCarrier.Data := _data.CarriersData[_i];
	
	IF _TemplateCarrier.HasWorkpiecesWithRequestStatus THEN
		HasCarrierWithRequestWorkpiece:= TRUE;
		RETURN;
	END_IF

END_FOR
END_GET
END_PROPERTY

{attribute 'monitoring' := 'call'}
PROPERTY PUBLIC HasCarrierWithUnfinishedWorkpiece : BOOL
GET
VAR
	_i : INT;
END_VAR
HasCarrierWithUnfinishedWorkpiece:= FALSE;
	
FOR _i:= 0 TO MAX_CARRIERPLACES DO

	THIS^._TemplateCarrier.Data := _data.CarriersData[_i];
	
	IF _TemplateCarrier.HasUnfinishedWorkpieces THEN
		HasCarrierWithUnfinishedWorkpiece:= TRUE;
		RETURN;
	END_IF

END_FOR
END_GET
END_PROPERTY

{attribute 'monitoring' := 'call'}
PROPERTY PUBLIC HasEmptySlot : BOOL
GET
VAR
	_i : INT;
END_VAR
HasEmptySlot:= FALSE;
	
FOR _i:= 0 TO MAX_CARRIERPLACES DO

	THIS^._TemplateCarrier.Data := _data.CarriersData[_i];
	
	IF NOT _TemplateCarrier.CarrierPresent THEN
		HasEmptySlot:= TRUE;
		RETURN;
	END_IF

END_FOR
END_GET
END_PROPERTY

PROPERTY InitialStatus : eTcaWorkpieceStatus
GET
InitialStatus := _config.CarrierConfig.InitialStatus;
END_GET
SET
VAR
	_i : INT;
END_VAR
_config.CarrierConfig.InitialStatus := InitialStatus;
END_SET
END_PROPERTY

METHOD PUBLIC IsEmptySlotAt : BOOL
VAR_INPUT
	Position	 : INT;
END_VAR
IF Position < 0 OR Position > MAX_CARRIERPLACES OR NOT _data.CarriersEnabled[Position] THEN
   IsEmptySlotAt := FALSE;
   RETURN;
END_IF
   
IsEmptySlotAt := NOT _data.CarriersData[Position].Enabled;
END_METHOD

METHOD PUBLIC RemoveCarrierAt : BOOL
VAR_INPUT
	Position	: INT;
END_VAR
IF Position < 0 OR Position > MAX_CARRIERPLACES OR NOT _data.CarriersEnabled[Position] THEN
   RETURN;
END_IF

_data.CarriersData[Position].Enabled := FALSE;
END_METHOD

PROPERTY RequestStatus : eTcaWorkpieceStatus
GET
RequestStatus := _config.CarrierConfig.RequestStatus;
END_GET
SET
_config.CarrierConfig.RequestStatus := RequestStatus;
END_SET
END_PROPERTY

{warning 'Methodenimplementierung hinzufügen'}
(*~
	<docu>
		<summary>
		    Custom service (manual, maintenance) logic.
			This method must be implemented in derived class.
		</summary>			
	</docu>	
~*)
METHOD ServiceMode
IF _service.DisableCarriers THEN 
_service.DisableCarriers := FALSE;
DisableCarriers(); 
END_IF

IF _service.EnableCarriers THEN 
_service.EnableCarriers := FALSE;
EnableCarriers(); 
END_IF

IF _service.FillWithEmptyCarriers THEN 
_service.FillWithEmptyCarriers := FALSE;
FillWithEmptyCarriers(); 
END_IF

IF _service.FillWithFinishedCarriers THEN 
_service.FillWithFinishedCarriers := FALSE;
FIllWithFinishedCarriers(); 
END_IF

IF _service.FillWithInitialCarriers THEN 
_service.FillWithInitialCarriers := FALSE;
FillWithInitialCarriers(); 
END_IF
END_METHOD

METHOD PUBLIC SetCarrierAt : BOOL
VAR_INPUT
	Position	: INT;
	Data : TcaCarrierData;
END_VAR
IF Position < 0 OR Position > MAX_CARRIERPLACES OR NOT _data.CarriersEnabled[Position] THEN
   RETURN;
END_IF

_data.CarriersData[Position]:= Data;
_data.CarriersData[Position].Enabled := TRUE;
END_METHOD

METHOD PUBLIC SetEmptyCarrierAt : BOOL
VAR_INPUT
	Position	: INT;
END_VAR
IF Position < 0 OR Position > MAX_CARRIERPLACES OR NOT _data.CarriersEnabled[Position] THEN
   RETURN;
END_IF

_TemplateCarrier.Config := _config.CarrierConfig;
_TemplateCarrier.EmptyCarrier();

_data.CarriersData[Position]:= _TemplateCarrier.Data;
_data.CarriersData[Position].Enabled := TRUE;
END_METHOD

METHOD PUBLIC SetFinishedCarrierAt : BOOL
VAR_INPUT
	Position	: INT;
END_VAR
IF Position < 0 OR Position > MAX_CARRIERPLACES OR NOT _data.CarriersEnabled[Position] THEN
   RETURN;
END_IF

_TemplateCarrier.Config := _config.CarrierConfig;
_TemplateCarrier.FinishCarrier();

_data.CarriersData[Position]:= _TemplateCarrier.Data;
_data.CarriersData[Position].Enabled := TRUE;
END_METHOD

METHOD PUBLIC SetInitialCarriersAt : BOOL
VAR_INPUT
	Position	: INT;
END_VAR
IF Position < 0 OR Position > MAX_CARRIERPLACES OR NOT _data.CarriersEnabled[Position] THEN
   RETURN;
END_IF

_TemplateCarrier.Config := _config.CarrierConfig;
_TemplateCarrier.InitialCarrier();

_data.CarriersData[Position]:= _TemplateCarrier.Data;
_data.CarriersData[Position].Enabled := TRUE;
END_METHOD

PROPERTY SlotOfCarrierWithEmptyWorkpieceplace : INT
GET
VAR
	_i : INT;
END_VAR
SlotOfCarrierWithEmptyWorkpieceplace:= -1;
	
FOR _i:= 0 TO MAX_CARRIERPLACES DO

	THIS^._TemplateCarrier.Data := _data.CarriersData[_i];
	
	IF _TemplateCarrier.HasEmptyWorkpieceplaces THEN
		SlotOfCarrierWithEmptyWorkpieceplace:= _i;
		RETURN;
	END_IF

END_FOR
END_GET
END_PROPERTY

PROPERTY SlotOfCarrierWithUnfinishedWorkpiece : INT
GET
VAR
	_i : INT;
END_VAR
SlotOfCarrierWithUnfinishedWorkpiece:= -1;
	
FOR _i:= 0 TO MAX_CARRIERPLACES DO

	THIS^._TemplateCarrier.Data := _data.CarriersData[_i];
	
	IF _TemplateCarrier.HasUnfinishedWorkpieces THEN
		SlotOfCarrierWithUnfinishedWorkpiece:= _i;
		RETURN;
	END_IF

END_FOR
END_GET
END_PROPERTY

{attribute 'monitoring' := 'call'}
PROPERTY PUBLIC TrolleyExists : BOOL
GET
TrolleyExists := _data.Exist;
END_GET
SET
_data.Exist := TrolleyExists;
END_SET
END_PROPERTY

END_FUNCTION_BLOCK

// ---- POUs/Items/TcaCarrier/TcaCarrier.TcPOU
FUNCTION_BLOCK TcaCarrier //EXTENDS TcoCore.TcoComponent  
VAR CONSTANT
	MAX_WORKPIECEPLACES : INT := 127;
END_VAR

VAR PERSISTENT
	_data : TcaCarrierData;
	_config : TcaCarrierConfig;
END_VAR

VAR	
	_WorkpiecesStatus : ARRAY[0..eTcaWorkpieceStatus.MAXSIZE] OF INT;
	_PrimaryStatus : eTcaWorkpieceStatus;
	_SecondaryStatus : eTcaWorkpieceStatus;
	_AllFinished : BOOL;
	_Unfinished : BOOL;
		
	_WorkpiecesCoordinate : ARRAY[0..TcaCarrier.MAX_WORKPIECEPLACES] OF ST_Coordinate;
	
END_VAR

RefreshStatus();

METHOD ApplyConfig
VAR
	tmpData				: TcaCarrierConfig;
	
	tmpOffset 			: REAL;
	tmpOddRow			: INT;
	tmpEvenRow			: INT;
	tmpWorkpieceCount	: INT;
	
	tmpPos		 		: INT;
	tmpLoc		 		: INT;		
	tmpRow 				: INT;
	//tmpLvl				: INT;
	
	nRowNumber			: INT;
	nLocationNumber		: INT; 
	
	ni					: INT;
	
	tmpCoordinate 		: ST_Coordinate;		
END_VAR
tmpData := _config;

//todo Error
//_ConfigError


CASE tmpData.Layout OF
	eTcaCarrierLayout.Layout1 : 
		tmpOffset := 0;
		tmpOddRow := tmpData.PositionsInRow;
	tmpEvenRow := tmpData.PositionsInRow;
        tmpWorkpieceCount := tmpData.PositionsInRow*tmpData.PositionsInColumn;
		
    eTcaCarrierLayout.Layout2 :
		tmpOffset := 0.5;
		tmpOddRow := tmpData.PositionsInRow;
		tmpEvenRow :=tmpData.PositionsInRow;
        tmpWorkpieceCount := tmpData.PositionsInRow*tmpData.PositionsInColumn;
		 
    eTcaCarrierLayout.Layout3 :
		 tmpOffset := -0.5;
		 tmpOddRow := tmpData.PositionsInRow;
         tmpEvenRow := tmpData.PositionsInRow;
         tmpWorkpieceCount := tmpData.PositionsInRow*tmpData.PositionsInColumn;	
		 
	eTcaCarrierLayout.Layout4 :
		 tmpOffset := -0.5;
		 tmpOddRow := tmpData.PositionsInRow;
         tmpEvenRow := tmpData.PositionsInRow + 1;
         tmpWorkpieceCount := tmpData.PositionsInRow*tmpData.PositionsInColumn + tmpData.PositionsInColumn/2;
		
	eTcaCarrierLayout.Layout5 :
		 tmpOffset := 0.5;
		 tmpOddRow := tmpData.PositionsInRow;
         tmpEvenRow := tmpData.PositionsInRow - 1;
         tmpWorkpieceCount := tmpData.PositionsInRow*tmpData.PositionsInColumn - tmpData.PositionsInColumn/2 - 1;
		 
END_CASE


MEMSET(ADR(_WorkpiecesCoordinate),0,SIZEOF(_WorkpiecesCoordinate));
MEMSET(ADR(_data.WorkpiecesEnabled),0,SIZEOF(_data.WorkpiecesEnabled));
//MEMSET(ADR(_data.WorkpiecesData),0,SIZEOF(_data.WorkpiecesData));


FOR ni:= 0 TO tmpWorkpieceCount-1 DO
	
	// Bestimmen des Reihen und Spaltenndex und der x und y-Koordinate
	tmpPos := ni MOD tmpWorkpieceCount;
	tmpRow := tmpPos/(tmpOddRow + tmpEvenRow);	
	tmpLoc := tmpPos MOD (tmpOddRow + tmpEvenRow);
	
	IF tmpLoc >= tmpOddRow THEN
	    // gerade Reihe
	    nRowNumber := tmpRow*2 + 1;
	    nLocationNumber := tmpLoc - tmpOddRow;
	    tmpCoordinate.fX := tmpData.ColumnDistance*(nLocationNumber + tmpOffset)+tmpData.CoordinateFirstWorkpiece.fX;
	    tmpCoordinate.fY := tmpData.RowDistance*nRowNumber+tmpData.CoordinateFirstWorkpiece.fY;
	ELSE
	    // ungerade Reihe
	    nRowNumber := tmpRow*2;
	    nLocationNumber := tmpLoc;
	    tmpCoordinate.fX := tmpData.ColumnDistance*nLocationNumber+tmpData.CoordinateFirstWorkpiece.fX;
	    tmpCoordinate.fY := tmpData.RowDistance*nRowNumber+tmpData.CoordinateFirstWorkpiece.fY;
	END_IF
	
	//tmpCoordinate.nOriginId := 0;
		
	_WorkpiecesCoordinate[ni] := tmpCoordinate;
	_data.WorkpiecesEnabled[ni] := TRUE;
	_data.Error := FALSE;

END_FOR
END_METHOD

{attribute 'monitoring' := 'call'}
PROPERTY PUBLIC CarrierPresent : BOOL
GET
CarrierPresent := _data.Enabled;
END_GET
END_PROPERTY

METHOD ColumnDistance : REFERENCE TO TcaCarrier
VAR_INPUT
	inDistance : LREAL;
END_VAR
THIS^._config.ColumnDistance:= inDistance;
ColumnDistance REF= THIS^;
END_METHOD

PROPERTY Config : REFERENCE TO TcaCarrierConfig
GET
Config REF= _config;
END_GET
SET
_config := Config;
END_SET
END_PROPERTY

METHOD CoordinateFirstWorkpiece : REFERENCE TO TcaCarrier
VAR_INPUT
	inCoordinate : ST_Coordinate;
END_VAR
THIS^._config.CoordinateFirstWorkpiece:= inCoordinate;
CoordinateFirstWorkpiece REF= THIS^;
END_METHOD

METHOD CoordinatesOf : ST_Coordinate
VAR_INPUT
	WorkpiecePlace		: INT;
END_VAR

VAR
	tmpData				: TcaCarrierConfig;
	
	tmpOffset 			: REAL;
	tmpOddRow			: INT;
	tmpEvenRow			: INT;
	tmpWorkpieceCount	: INT;
	
	tmpPos		 		: INT;
	tmpLoc		 		: INT;		
	tmpRow 				: INT;
	//tmpLvl				: INT;
	
	nRowNumber			: INT;
	nLocationNumber		: INT; 
	
	tmpCoordinate 		: ST_Coordinate;		
	
END_VAR
IF NOT _data.WorkpiecesEnabled[WorkpiecePlace] THEN
	RETURN;
END_IF	

CoordinatesOf := _WorkpiecesCoordinate[WorkpiecePlace];
END_METHOD

METHOD CountEmptyPlaces : INT

VAR
	tmp				: INT;
	ni				: INT;
END_VAR
CountEmptyPlaces := CountPlacesByStatus(eTcaWorkpieceStatus.undefined);
END_METHOD

METHOD CountPlacesByStatus : INT
VAR_INPUT
	Status			: eTcaWorkpieceStatus;
END_VAR

VAR
	tmp				: INT;
	ni				: INT;
END_VAR
CountPlacesByStatus := 0;

FOR ni := 0 TO MAX_WORKPIECEPLACES DO

	IF NOT _data.WorkpiecesEnabled[ni] THEN
		CONTINUE;
	END_IF	
	
	IF _data.WorkpiecesData[ni].Error THEN
		CONTINUE;
	END_IF

	IF _data.WorkpiecesData[ni].CurrentStatus = Status THEN
			tmp := tmp + 1;
	END_IF
	
END_FOR

CountPlacesByStatus := tmp;
END_METHOD

PROPERTY Data : REFERENCE TO TcaCarrierData
GET
Data REF= _data;
END_GET
SET
_data := Data;
RefreshStatus();
END_SET
END_PROPERTY

{attribute 'TcRpcEnable'}
METHOD EmptyCarrier : TcaCarrierData
VAR
	_i			: INT;
END_VAR
_data.Enabled := TRUE;
	
FOR _i := 0 TO MAX_WORKPIECEPLACES DO	
	
	IF NOT _data.WorkpiecesEnabled[_i] THEN
		RETURN;
	END_IF	

	_data.WorkpiecesData[_i].Error := FALSE;
	_data.WorkpiecesData[_i].Logging := "";	// TIMESTAMP WIT MESSAGE
	_data.WorkpiecesData[_i].SerialNumber := '';
	_data.WorkpiecesData[_i].CurrentStatus := eTcaWorkpieceStatus.undefined;	
	_data.WorkpiecesData[_i].InitialStatus := _config.InitialStatus;
	_data.WorkpiecesData[_i].RequestStatus := _config.RequestStatus;
	
END_FOR
END_METHOD

METHOD FindPlace : REFERENCE TO TcaWorkpieceData //-1..no Position found

VAR_INPUT
	Status		: eTcaWorkpieceStatus;
END_VAR

VAR
	ni				: INT;
END_VAR
FindPlace REF= 0;
FOR ni := 0 TO MAX_WORKPIECEPLACES DO
	
	IF NOT _data.WorkpiecesEnabled[ni] THEN
		CONTINUE;
	END_IF	
	
	IF _data.WorkpiecesData[ni].Error THEN
		CONTINUE;
	END_IF	

	IF _data.WorkpiecesData[ni].CurrentStatus = Status OR Status < eTcaWorkpieceStatus.undefined THEN	   
		FindPlace REF= _data.WorkpiecesData[ni];		
	END_IF	
END_FOR
END_METHOD

{attribute 'TcRpcEnable'}
METHOD FinishCarrier : TcaCarrierData
VAR
	_i			: INT;
END_VAR
_data.Enabled := TRUE;
	
FOR _i := 0 TO MAX_WORKPIECEPLACES DO	
	
	IF NOT _data.WorkpiecesEnabled[_i] THEN
		RETURN;
	END_IF	

	_data.WorkpiecesData[_i].Error := FALSE;
	_data.WorkpiecesData[_i].Logging := "";	// TIMESTAMP WIT MESSAGE
	_data.WorkpiecesData[_i].SerialNumber := '';
	_data.WorkpiecesData[_i].CurrentStatus := config.RequestStatus;	
	_data.WorkpiecesData[_i].InitialStatus := _config.InitialStatus;
	_data.WorkpiecesData[_i].RequestStatus := _config.RequestStatus;
	
END_FOR
END_METHOD

METHOD GetPlaceReference : REFERENCE TO TcaWorkpieceData
VAR_INPUT
	IndexNr		: INT;
END_VAR
IF IndexNr < 0 OR IndexNr > MAX_WORKPIECEPLACES THEN
	RETURN;
END_IF

GetPlaceReference REF= _data.WorkpiecesData[IndexNr];
END_METHOD

{attribute 'monitoring' := 'call'}
PROPERTY PUBLIC HasAllWorkpiecesFinished : BOOL
GET
HasAllWorkpiecesFinished := _AllFinished;
END_GET
END_PROPERTY

{attribute 'monitoring' := 'call'}
PROPERTY PUBLIC HasEmptyWorkpieceplaces : BOOL
GET
HasEmptyWorkpieceplaces := CountEmptyPlaces() > 0;
END_GET
END_PROPERTY

{attribute 'monitoring' := 'call'}
PROPERTY PUBLIC HasUnfinishedWorkpieces : BOOL
GET
HasUnfinishedWorkpieces := _Unfinished;
END_GET
END_PROPERTY

{attribute 'monitoring' := 'call'}
PROPERTY PUBLIC HasWorkpiecesWithInitialStatus : BOOL
GET
HasWorkpiecesWithInitialStatus := CountPlacesByStatus(_config.InitialStatus) > 0;
END_GET
END_PROPERTY

{attribute 'monitoring' := 'call'}
PROPERTY PUBLIC HasWorkpiecesWithRequestStatus : BOOL
GET
HasWorkpiecesWithRequestStatus := CountPlacesByStatus(_config.RequestStatus) > 0;
END_GET
END_PROPERTY

{attribute 'TcRpcEnable'}
METHOD InitialCarrier : TcaCarrierData
VAR
	_i			: INT;
END_VAR

VAR_INST
	WorkpieceCtrl : TcaWorkpieceControl;//(This^);
END_VAR
_data.Enabled := TRUE;

FOR _i := 0 TO MAX_WORKPIECEPLACES DO	
	
	IF NOT _data.WorkpiecesEnabled[_i] THEN
		RETURN;
	END_IF	

	_data.WorkpiecesData[_i].Id := _i+1;
	_data.WorkpiecesData[_i].Error := FALSE;
	_data.WorkpiecesData[_i].SerialNumber := '';
	_data.WorkpiecesData[_i].CurrentStatus := _config.InitialStatus;	
	_data.WorkpiecesData[_i].InitialStatus := _config.InitialStatus;
	_data.WorkpiecesData[_i].RequestStatus := _config.RequestStatus;
	
	WorkpieceCtrl.SetReference(_data.WorkpiecesData[_i]);
	WorkpieceCtrl.LogEntry('New Workpiece');
	
	
END_FOR
END_METHOD

PROPERTY InitialStatus : eTcaWorkpieceStatus
GET
InitialStatus := _config.InitialStatus;
END_GET
SET
_config.InitialStatus := InitialStatus;
END_SET
END_PROPERTY

METHOD Layout : REFERENCE TO TcaCarrier
VAR_INPUT
	inLayout : eTcaCarrierLayout;
END_VAR
THIS^._config.Layout:= inLayout;
Layout REF= THIS^;
END_METHOD

METHOD PositionsInColumn : REFERENCE TO TcaCarrier
VAR_INPUT
	inPositionsInColumn : INT;
END_VAR
THIS^._config.PositionsInColumn:= inPositionsInColumn;
PositionsInColumn REF= THIS^;
END_METHOD

METHOD PositionsInRow : REFERENCE TO TcaCarrier
VAR_INPUT
	inPositionsInRow : INT;
END_VAR
THIS^._config.PositionsInRow:= inPositionsInRow;
PositionsInRow REF= THIS^;
END_METHOD

METHOD RefreshStatus : BOOL
VAR
	ni			: INT;
END_VAR
MEMSET(ADR(_WorkpiecesStatus), 0, SIZEOF(_WorkpiecesStatus));

_PrimaryStatus := eTcaWorkpieceStatus.undefined;
_SecondaryStatus := eTcaWorkpieceStatus.undefined;
_AllFinished := _data.Enabled;
_UnFinished := FALSE;

FOR ni := 0 TO MAX_WORKPIECEPLACES DO
	
	IF NOT _data.WorkpiecesEnabled[ni] THEN
		CONTINUE;
	END_IF
	
	IF _data.WorkpiecesData[ni].Exist AND
	   NOT _data.WorkpiecesData[ni].Error AND
       NOT _data.WorkpiecesData[ni].CurrentStatus <> _data.WorkpiecesData[ni].RequestStatus THEN
		_AllFinished := FALSE;
		_UnFinished := TRUE;
	END_IF
	
	_WorkpiecesStatus[_data.WorkpiecesData[ni].CurrentStatus] := _WorkpiecesStatus[_data.WorkpiecesData[ni].CurrentStatus] + 1;
	
	IF _WorkpiecesStatus[_data.WorkpiecesData[ni].CurrentStatus] >= _WorkpiecesStatus[_PrimaryStatus] THEN
		_SecondaryStatus := _PrimaryStatus;
		_PrimaryStatus := _data.WorkpiecesData[ni].CurrentStatus;
	END_IF

END_FOR


IF _PrimaryStatus = _SecondaryStatus THEN
	_SecondaryStatus := eTcaWorkpieceStatus.undefined;
END_IF
END_METHOD

{attribute 'TcRpcEnable'}
METHOD RemoveCarrier : TcaCarrierData
VAR
	_i			: INT;
END_VAR
_data.Enabled := FALSE;
END_METHOD

PROPERTY RequestStatus : eTcaWorkpieceStatus
GET
RequestStatus := _config.RequestStatus;
END_GET
SET
_config.RequestStatus := RequestStatus;
END_SET
END_PROPERTY

METHOD RowDistance : REFERENCE TO TcaCarrier
VAR_INPUT
	inDistance : LREAL;
END_VAR
THIS^._config.RowDistance:= inDistance;
RowDistance REF= THIS^;
END_METHOD

{attribute 'TcRpcEnable'}
METHOD SetCarrier : TcaCarrierData
VAR_INPUT
	Data	: TcaCarrierData;
	//Source	: E_Station;
END_VAR
_data := Data;
_data.Enabled := TRUE;
//_data.Source := Source;
END_METHOD

PROPERTY WorkpiecePlaces : INT
GET
CASE _config.Layout OF	
	eTcaCarrierLayout.Layout1 : WorkpiecePlaces := _config.PositionsInRow*_config.PositionsInColumn;		
    eTcaCarrierLayout.Layout2 : WorkpiecePlaces := _config.PositionsInRow*_config.PositionsInColumn;		 
    eTcaCarrierLayout.Layout3 : WorkpiecePlaces := _config.PositionsInRow*_config.PositionsInColumn;		 
	eTcaCarrierLayout.Layout4 : WorkpiecePlaces := _config.PositionsInRow*_config.PositionsInColumn + _config.PositionsInColumn/2;		
	eTcaCarrierLayout.Layout5 : WorkpiecePlaces := _config.PositionsInRow*_config.PositionsInColumn - _config.PositionsInColumn/2;		
	ELSE
		 WorkpiecePlaces := 0;
END_CASE
END_GET
END_PROPERTY

PROPERTY WorkpiecesStatusCount : ARRAY[0..eTcaWorkpieceStatus.MAXSIZE] OF INT
GET
WorkpiecesStatusCount := _WorkpiecesStatus;
END_GET
END_PROPERTY

END_FUNCTION_BLOCK

// ---- POUs/Items/TcaWorkpiece/TcaWorkpieceControl.TcPOU
FUNCTION_BLOCK TcaWorkpieceControl //EXTENDS TcoComponent

VAR
	_data	: REFERENCE TO TcaWorkpieceData;
END_VAR

IF NOT __ISVALIDREF(_data) THEN
	RETURN;
END_IF

METHOD LogEntry : STRING;
VAR_INPUT
	Message : STRING;
END_VAR

VAR
	tmpString		: STRING;
END_VAR
IF NOT __ISVALIDREF(_data) THEN
	RETURN;
END_IF

tmpString := concat(tmpString, DT_TO_STRING(Statics.dtNow));
tmpString := concat(tmpString, ' | ');
tmpString := concat(tmpString, Message);
tmpString := Concat(tmpString, '$N');
_data.Logging:=  TO_WSTRING(tmpString);

LogEntry := tmpString;
END_METHOD

{warning 'Methodenimplementierung hinzufügen'}
(*~
	<docu>
		<summary>
		    Custom service (manual, maintenance) logic.
			This method must be implemented in derived class.
		</summary>			
	</docu>	
~*)
METHOD PROTECTED ServiceMode
END_METHOD

METHOD INTERNAL SetEmpty : REFERENCE TO TcaWorkpieceControl
VAR
END_VAR
IF NOT __ISVALIDREF(_data) THEN
	RETURN;
END_IF

SetEmpty REF= THIS^;

_data.CurrentStatus := eTcaWorkpieceStatus.undefined;
_data.InitialStatus := eTcaWorkpieceStatus.undefined;
_data.RequestStatus := eTcaWorkpieceStatus.undefined;

_data.Logging:= "";
_data.SerialNumber := '';
_data.TimeStampChanged := Statics.dtNow;
_data.Error := FALSE;
_data.Exist := FALSE;
END_METHOD

METHOD INTERNAL SetReference : REFERENCE TO TcaWorkpieceControl
VAR_IN_OUT
	Data : TcaWorkpieceData;
END_VAR
_Data REF= Data;

SetReference REF= THIS^;
END_METHOD

METHOD INTERNAL SetWorkpiece : REFERENCE TO TcaWorkpieceControl
VAR
	InitialStatus	: eTcaWorkpieceStatus;
	RequestStatus	: eTcaWorkpieceStatus;
END_VAR
IF NOT __ISVALIDREF(_data) THEN
	RETURN;
END_IF

SetWorkpiece REF= THIS^;

_data.CurrentStatus := InitialStatus;
_data.InitialStatus := InitialStatus;
_data.RequestStatus := RequestStatus;

_data.Exist := TRUE;
_data.TimeStampChanged := Statics.dtNow;
LogEntry('New Workpiece');
END_METHOD

END_FUNCTION_BLOCK

// ---- POUs/Plant/ST030_Handling/FB_St030_Handling.TcPOU
FUNCTION_BLOCK FB_St030_Handling EXTENDS FB_StationBase
VAR_INPUT
END_VAR
VAR	
	// IO ref
	stIO			: REFERENCE TO ST_St030_IO;
	
	// station components
	fbAxisX 		: FB_AxisDriver;
	fbAxisY 		: FB_AxisDriver;
	fbAxisZ 		: FB_AxisDriver;
	
	// actor UIs, access to: iStatus, fPosition, iVisibleState, ..
	fbAxisXUi		: FB_Axis_Ui;
	fbAxisYUi		: FB_Axis_Ui;
	fbAxisZUi		: FB_Axis_Ui;
	
	// instance var's
	bStationDeaktiv	: BOOL;
	
	eEmptyChk		: E_St030_EmptySlotChk;
	sqSearch		: FB_SequenceHelperSb;
	fPosSearchCorr	: LREAL;
	SearchTrig		: ARRAY[0..1, 0..1] OF ST_XZ_Point; // S1/S2 - Trig 1/2
	fThreshMesMin	: LREAL := 320;
	fThreshMesMax	: LREAL := 350;
END_VAR
VAR PERSISTENT
	HgPosBackup		: ST_3DPoint;
END_VAR

/// 
/// Station 030 function block - Handling
///

METHOD PRIVATE GetPosOvRp : LREAL
VAR_INPUT
	iOven,					// oven 1/2 (A/B)
	iRp		: INT;			// ref point 1/2
	sAxis	: STRING(1); 	// axis X/Y/Z
END_VAR
VAR
	ovRp	: INT;
END_VAR
// get reference point value for specified oven, point and axis

ovRp := (iOven * 10) + iRp;
CASE ovRp OF
	 11:
		IF sAxis = 'X' THEN
			GetPosOvRp := stSettings.stStationSettings[E_Station.eStation_ST010_OvenA].stDynStationSettings[E_St010_Settings.eSt010_Settings_XPosRp1].fValue;
		ELSIF sAxis = 'Y' THEN                                                                      
			GetPosOvRp := stSettings.stStationSettings[E_Station.eStation_ST010_OvenA].stDynStationSettings[E_St010_Settings.eSt010_Settings_YPosRp1].fValue;
		ELSIF sAxis = 'Z' THEN                                                                      
			GetPosOvRp := stSettings.stStationSettings[E_Station.eStation_ST010_OvenA].stDynStationSettings[E_St010_Settings.eSt010_Settings_ZPosRp1].fValue;
		END_IF                                                                                      
		                                                                                            
	12:                                                                                             
		IF sAxis = 'X' THEN                                                                         
			GetPosOvRp := stSettings.stStationSettings[E_Station.eStation_ST010_OvenA].stDynStationSettings[E_St010_Settings.eSt010_Settings_XPosRp2].fValue;
		ELSIF sAxis = 'Y' THEN                                                                      
			GetPosOvRp := stSettings.stStationSettings[E_Station.eStation_ST010_OvenA].stDynStationSettings[E_St010_Settings.eSt010_Settings_YPosRp2].fValue;
		ELSIF sAxis = 'Z' THEN                                                                      
			GetPosOvRp := stSettings.stStationSettings[E_Station.eStation_ST010_OvenA].stDynStationSettings[E_St010_Settings.eSt010_Settings_ZPosRp2].fValue;
		END_IF                                                                                      
		                                                                                            
	21:                                                                                             
		IF sAxis = 'X' THEN                                                                         
			GetPosOvRp := stSettings.stStationSettings[E_Station.eStation_ST020_OvenB].stDynStationSettings[E_St020_Settings.eSt020_Settings_XPosRp1].fValue;
		ELSIF sAxis = 'Y' THEN                                                                      
			GetPosOvRp := stSettings.stStationSettings[E_Station.eStation_ST020_OvenB].stDynStationSettings[E_St020_Settings.eSt020_Settings_YPosRp1].fValue;
		ELSIF sAxis = 'Z' THEN                                                                      
			GetPosOvRp := stSettings.stStationSettings[E_Station.eStation_ST020_OvenB].stDynStationSettings[E_St020_Settings.eSt020_Settings_ZPosRp1].fValue;
		END_IF                                                                                      
		                                                                                            
	22:                                                                                             
		IF sAxis = 'X' THEN                                                                         
			GetPosOvRp := stSettings.stStationSettings[E_Station.eStation_ST020_OvenB].stDynStationSettings[E_St020_Settings.eSt020_Settings_XPosRp2].fValue;
		ELSIF sAxis = 'Y' THEN                                                                      
			GetPosOvRp := stSettings.stStationSettings[E_Station.eStation_ST020_OvenB].stDynStationSettings[E_St020_Settings.eSt020_Settings_YPosRp2].fValue;
		ELSIF sAxis = 'Z' THEN                                                                      
			GetPosOvRp := stSettings.stStationSettings[E_Station.eStation_ST020_OvenB].stDynStationSettings[E_St020_Settings.eSt020_Settings_ZPosRp2].fValue;
		END_IF
END_CASE
END_METHOD

{attribute 'monitoring' := 'call'}
PROPERTY INTERNAL HgRefPosX : LREAL
GET
HgRefPosX := stLocalSettings.stDynStationSettings[E_St030_Settings.eSt030_Settings_AxisRefPosX].fValue;
END_GET
END_PROPERTY

{attribute 'monitoring' := 'call'}
PROPERTY INTERNAL HgRefPosY : LREAL
GET
HgRefPosY := stLocalSettings.stDynStationSettings[E_St030_Settings.eSt030_Settings_AxisRefPosY].fValue;
END_GET
END_PROPERTY

{attribute 'monitoring' := 'call'}
PROPERTY INTERNAL HgRefPosZ : LREAL
GET
HgRefPosZ := stLocalSettings.stDynStationSettings[E_St030_Settings.eSt030_Settings_AxisRefPosZ].fValue;
END_GET
END_PROPERTY

{attribute 'monitoring' := 'call'}
PROPERTY PRIVATE HomeSpeedX : LREAL
GET
HomeSpeedX := stLocalSettings.stDynStationSettings[E_St030_Settings.eSt030_Settings_XHomeSpeed].fValue;
END_GET
END_PROPERTY

{attribute 'monitoring' := 'call'}
PROPERTY PRIVATE HomeSpeedY : LREAL
GET
HomeSpeedY := stLocalSettings.stDynStationSettings[E_St030_Settings.eSt030_Settings_YHomeSpeed].fValue;
END_GET
END_PROPERTY

